  MoveL 2042 to (226.09, 430.21, -17.52) mm, rotated rx -180 ry 0 rz -11.91 deg; joints [26.659, -20.064, 61.919, -79.673, 100.73, 132.011]
  MoveL 2043 to (226.02, 430.34, -17.52) mm, rotated rx 180 ry 0 rz -11.91 deg; joints [26.655, -20.058, 61.906, -79.677, 100.728, 132.004]
  MoveL 2044 to (225.94, 430.47, -17.53) mm, rotated rx -180 ry 0 rz -11.91 deg; joints [26.652, -20.052, 61.893, -79.681, 100.727, 131.996]
  MoveL 2045 to (225.78, 430.71, -17.53) mm, rotated rx 180 ry 0 rz -11.91 deg; joints [26.644, -20.041, 61.871, -79.689, 100.723, 131.983]
  MoveL 2046 to (225.58, 430.96, -17.53) mm, rotated rx 180 ry 0 rz -11.91 deg; joints [26.635, -20.032, 61.851, -79.697, 100.718, 131.972]
  MoveL 2047 to (225.44, 431.1, -17.52) mm, rotated rx -180 ry 0 rz -11.91 deg; joints [26.629, -20.027, 61.84, -79.702, 100.715, 131.966]
  MoveL 2048 to (225.3, 431.23, -17.53) mm, rotated rx -180 ry 0 rz -11.91 deg; joints [26.623, -20.023, 61.833, -79.706, 100.712, 131.961]
  MoveL 2049 to (225.16, 431.34, -17.53) mm, rotated rx -180 ry 0 rz -11.91 deg; joints [26.618, -20.02, 61.827, -79.711, 100.708, 131.957]
  MoveL 2050 to (225.02, 431.44, -17.53) mm, rotated rx -180 ry 0 rz -11.91 deg; joints [26.612, -20.018, 61.822, -79.715, 100.705, 131.954]
  MoveL 2051 to (224.78, 431.59, -17.52) mm, rotated rx -180 ry 0 rz -11.91 deg; joints [26.604, -20.016, 61.818, -79.721, 100.699, 131.951]
  MoveL 2052 to (224.55, 431.71, -17.53) mm, rotated rx -180 ry 0 rz -11.91 deg; joints [26.596, -20.016, 61.818, -79.727, 100.693, 131.95]
  MoveL 2053 to (224.32, 431.8, -17.53) mm, rotated rx -180 ry 0 rz -11.91 deg; joints [26.588, -20.017, 61.821, -79.732, 100.687, 131.951]
  MoveL 2054 to (224.09, 431.88, -17.53) mm, rotated rx -180 ry 0 rz -11.91 deg; joints [26.581, -20.02, 61.827, -79.736, 100.681, 131.953]
  MoveL 2055 to (224.01, 431.9, -17.53) mm, rotated rx -180 ry 0 rz -11.91 deg; joints [26.579, -20.021, 61.829, -79.738, 100.679, 131.954]
  MoveL 2056 to (223.77, 431.95, -17.53) mm, rotated rx -180 ry 0 rz -11.91 deg; joints [26.571, -20.025, 61.839, -79.742, 100.673, 131.958]
  MoveL 2057 to (223.53, 431.98, -17.53) mm, rotated rx -180 ry 0 rz -11.91 deg; joints [26.564, -20.031, 61.851, -79.745, 100.666, 131.963]
  MoveL 2058 to (223.29, 431.99, -17.53) mm, rotated rx -180 ry 0 rz -11.91 deg; joints [26.557, -20.038, 61.866, -79.749, 100.66, 131.97]
  MoveL 2059 to (223.05, 431.99, -17.53) mm, rotated rx -180 ry 0 rz -11.91 deg; joints [26.551, -20.046, 61.883, -79.752, 100.653, 131.978]
  MoveL 2060 to (-164.9, 431.99, -17.52) mm, rotated rx -180 ry 0 rz -11.91 deg; joints [14.903, -28.534, 80.361, -87.324, 91.595, 141.007]
  MoveL 2061 to (-194.97, 431.99, -17.53) mm, rotated rx 180 ry 0 rz -11.91 deg; joints [13.93, -28.928, 81.241, -88.082, 90.978, 141.468]
  MoveL 2062 to (-195.47, 431.99, -17.53) mm, rotated rx 180 ry 0 rz -11.91 deg; joints [13.914, -28.934, 81.255, -88.094, 90.967, 141.475]
  Set speed (38.1 mm/s)
  MoveL 2063 to (-196.09, 432.77, -17.53) mm, rotated rx -180 ry 0 rz -11.91 deg; joints [13.888, -28.902, 81.184, -88.116, 90.952, 141.437]
  MoveL 2064 to (-195.65, 434.72, -17.52) mm, rotated rx 180 ry 0 rz -11.91 deg; joints [13.886, -28.795, 80.951, -88.119, 90.956, 141.311]
  MoveL 2065 to (-195.51, 435.34, -16.89) mm, rotated rx 180 ry 0 rz -11.91 deg; joints [13.886, -28.791, 80.884, -88.121, 90.957, 141.248]
  Set speed (100.0 mm/s)
  MoveL 2066 to (-195.51, 435.34, 34.52) mm, rotated rx 180 ry 0 rz -11.91 deg; joints [13.873, -31.158, 81.335, -88.164, 91.012, 139.332]
  MoveL 2067 to (-195.51, 435.34, 34.52) mm, rotated rx 180 ry 0 rz -11.91 deg; joints [13.873, -31.158, 81.335, -88.164, 91.012, 139.332]

--- program Machining (robot KUKA KR 30 HA) ---
  Smooth(15)
  Print: /'1001'
  Print: /''
  Print: /'Parallel1'
  Set speed (100.0 mm/s)
  Set Ref.: Frame 4
  Set Tool: rc90 spindle mm
  Show rc90 spindle mm
  MoveJ 1 to (194.72, 277.93, 99.72) mm, rotated rx -149.92 ry 0.28 rz 179.52 deg; joints [13.584, -45.402, 109.059, -165.249, 63.754, 203.812]
  MoveL 2 to (194.72, 277.93, 99.72) mm, rotated rx -149.92 ry 0.28 rz 179.52 deg; joints [13.584, -45.402, 109.059, -165.249, 63.754, 203.812]
  MoveL 3 to (194.72, 227.8, 13.19) mm, rotated rx -149.92 ry 0.28 rz 179.52 deg; joints [15.532, -40.122, 107.271, -163.55, 67.335, 203.986]
  MoveL 4 to (194.72, 227.8, 13.19) mm, rotated rx -149.92 ry 0.28 rz 179.52 deg; joints [15.532, -40.122, 107.271, -163.55, 67.335, 203.986]
  Set speed (100.0 mm/s)
  MoveL 5 to (194.72, 218.79, -2.36) mm, rotated rx -149.92 ry 0.28 rz 179.52 deg; joints [15.878, -39.152, 106.869, -163.244, 67.917, 204.023]
  Set speed (16.7 mm/s)
  MoveL 6 to (194.72, 209.92, -17.68) mm, rotated rx -149.92 ry 0.28 rz 179.52 deg; joints [16.219, -38.193, 106.45, -162.942, 68.471, 204.061]
  MoveL 7 to (193.72, 209.42, -18.55) mm, rotated rx -149.92 ry 0.28 rz 179.52 deg; joints [16.249, -38.173, 106.512, -162.919, 68.552, 204.075]
  MoveL 8 to (193.59, 214.43, -9.89) mm, rotated rx -149.92 ry 0.28 rz 179.52 deg; joints [16.058, -38.721, 106.764, -163.089, 68.248, 204.055]
  MoveL 9 to (193.59, 214.44, -9.88) mm, rotated rx -149.92 ry 0.28 rz 179.52 deg; joints [16.058, -38.722, 106.764, -163.089, 68.248, 204.055]
  Set speed (100.0 mm/s)
  MoveL 10 to (193.59, 222.79, 4.53) mm, rotated rx -149.92 ry 0.28 rz 179.52 deg; joints [15.737, -39.624, 107.148, -163.373, 67.718, 204.02]
  MoveL 11 to (194.72, 224.52, 3.53) mm, rotated rx -149.92 ry 0.28 rz 179.52 deg; joints [15.659, -39.543, 107.081, -163.458, 67.722, 204.054]
  MoveL 12 to (194.72, 217.03, -9.4) mm, rotated rx -149.92 ry 0.28 rz 179.52 deg; joints [15.947, -38.735, 106.737, -163.203, 68.198, 204.085]
  Set speed (16.7 mm/s)
  MoveL 13 to (194.72, 211.65, -18.68) mm, rotated rx -149.92 ry 0.28 rz 179.52 deg; joints [16.154, -38.152, 106.48, -163.02, 68.531, 204.108]
  MoveC 14 to (194.43, 211.3, -19.3) mm, rotated rx -149.92 ry 0.28 rz 179.52 deg; joints [16.17, -38.124, 106.488, -163.006, 68.568, 204.113] to (193.72, 211.15, -19.55) mm, rotated rx -149.92 ry 0.28 rz 179.52 deg; joints [16.184, -38.133, 106.542, -162.997, 68.613, 204.122]
  MoveL 15 to (193.72, 211.15, -19.55) mm, rotated rx -149.92 ry 0.28 rz 179.52 deg; joints [16.184, -38.133, 106.542, -162.997, 68.613, 204.122]
  MoveL 16 to (193.49, 216.16, -10.9) mm, rotated rx -149.92 ry 0.28 rz 179.52 deg; joints [15.994, -38.685, 106.803, -163.166, 68.314, 204.104]
  MoveL 17 to (191.2, 216.16, -10.9) mm, rotated rx -149.92 ry 0.28 rz 179.52 deg; joints [16.019, -38.765, 107.001, -163.153, 68.429, 204.131]
  MoveC 18 to (190.5, 216.31, -10.64) mm, rotated rx -149.92 ry 0.28 rz 179.52 deg; joints [16.021, -38.806, 107.069, -163.154, 68.455, 204.138] to (190.2, 216.66, -10.03) mm, rotated rx -149.92 ry 0.28 rz 179.52 deg; joints [16.011, -38.855, 107.111, -163.164, 68.448, 204.14]
  MoveL 19 to (190.2, 216.66, -10.03) mm, rotated rx -149.92 ry 0.28 rz 179.52 deg; joints [16.011, -38.855, 107.111, -163.164, 68.448, 204.14]
  Set speed (100.0 mm/s)
  MoveL 20 to (190.2, 224.52, 3.53) mm, rotated rx -149.92 ry 0.28 rz 179.52 deg; joints [15.708, -39.705, 107.472, -163.432, 67.947, 204.106]
  MoveL 21 to (-191.54, 222.79, 4.53) mm, rotated rx -149.92 ry 0.28 rz 179.52 deg; joints [21.283, -50.457, 136.898, -159.048, 86.021, 209.028]
  MoveL 22 to (-191.54, 219.49, -1.15) mm, rotated rx -149.92 ry 0.28 rz 179.52 deg; joints [21.448, -49.971, 136.724, -158.89, 86.316, 209.131]
  Set speed (16.7 mm/s)
  MoveL 23 to (-191.54, 214.63, -9.56) mm, rotated rx -149.92 ry 0.28 rz 179.52 deg; joints [21.69, -49.254, 136.461, -158.658, 86.744, 209.284]
  MoveL 24 to (-191.93, 214.43, -9.89) mm, rotated rx -149.92 ry 0.28 rz 179.52 deg; joints [21.707, -49.232, 136.477, -158.641, 86.78, 209.297]
  MoveL 25 to (-192.68, 214.43, -9.89) mm, rotated rx -149.92 ry 0.28 rz 179.52 deg; joints [21.722, -49.246, 136.529, -158.627, 86.815, 209.31]
  MoveL 26 to (-192.7, 209.42, -18.55) mm, rotated rx -149.92 ry 0.28 rz 179.52 deg; joints [21.971, -48.509, 136.25, -158.387, 87.245, 209.468]
  MoveL 27 to (-193.07, 211.15, -19.55) mm, rotated rx -149.92 ry 0.28 rz 179.52 deg; joints [21.894, -48.445, 136.307, -158.465, 87.357, 209.515]
  MoveL 28 to (-193.07, 216.16, -10.9) mm, rotated rx -149.92 ry 0.28 rz 179.52 deg; joints [21.645, -49.182, 136.587, -158.707, 86.927, 209.358]
  MoveL 29 to (-189.43, 216.16, -10.9) mm, rotated rx -149.92 ry 0.28 rz 179.52 deg; joints [21.574, -49.115, 136.335, -158.774, 86.753, 209.294]
  MoveL 30 to (-188.93, 216.41, -10.46) mm, rotated rx -149.92 ry 0.28 rz 179.52 deg; joints [21.552, -49.143, 136.314, -158.795, 86.708, 209.277]
  MoveC 31 to (-189.34, 217.09, -9.63) mm, rotated rx -149.92 ry 0.28 rz 179.52 deg; joints [21.527, -49.223, 136.374, -158.82, 86.689, 209.271] to (-190.32, 217.64, -9.44) mm, rotated rx -149.92 ry 0.28 rz 179.52 deg; joints [21.519, -49.26, 136.461, -158.829, 86.735, 209.289]
  MoveL 32 to (-190.32, 217.64, -9.44) mm, rotated rx -149.92 ry 0.28 rz 179.52 deg; joints [21.519, -49.26, 136.461, -158.829, 86.735, 209.289]
  MoveL 33 to (-192.56, 218.42, -9.89) mm, rotated rx -149.92 ry 0.28 rz 179.52 deg; joints [21.525, -49.27, 136.63, -158.826, 86.884, 209.347]
  MoveC 34 to (-193.55, 218.53, -10.47) mm, rotated rx -149.92 ry 0.28 rz 179.52 deg; joints [21.538, -49.242, 136.692, -158.815, 86.968, 209.379] to (-193.96, 218.14, -11.47) mm, rotated rx -149.92 ry 0.28 rz 179.52 deg; joints [21.566, -49.165, 136.694, -158.788, 87.042, 209.406]
  MoveL 35 to (-193.96, 218.14, -11.47) mm, rotated rx -149.92 ry 0.28 rz 179.52 deg; joints [21.566, -49.165, 136.694, -158.788, 87.042, 209.406]
  MoveL 36 to (-193.96, 213.13, -20.12) mm, rotated rx -149.92 ry 0.28 rz 179.52 deg; joints [21.815, -48.426, 136.413, -158.546, 87.472, 209.564]
  MoveL 37 to (-193.46, 212.88, -20.55) mm, rotated rx -149.92 ry 0.28 rz 179.52 deg; joints [21.818, -48.381, 136.364, -158.544, 87.469, 209.563]
  MoveL 38 to (-193.43, 217.89, -11.9) mm, rotated rx -149.92 ry 0.28 rz 179.52 deg; joints [21.568, -49.118, 136.644, -158.786, 87.038, 209.405]
  MoveL 39 to (193.49, 217.89, -11.9) mm, rotated rx -149.92 ry 0.28 rz 179.52 deg; joints [15.929, -38.644, 106.833, -163.244, 68.375, 204.151]
  MoveL 40 to (193.72, 212.88, -20.55) mm, rotated rx -149.92 ry 0.28 rz 179.52 deg; joints [16.119, -38.092, 106.572, -163.074, 68.673, 204.169]
  MoveL 41 to (193.72, 214.61, -21.55) mm, rotated rx -149.92 ry 0.28 rz 179.52 deg; joints [16.054, -38.052, 106.601, -163.152, 68.733, 204.215]
  MoveL 42 to (193.49, 219.62, -12.9) mm, rotated rx -149.92 ry 0.28 rz 179.52 deg; joints [15.864, -38.604, 106.863, -163.322, 68.435, 204.197]
  MoveL 43 to (-193.72, 219.62, -12.9) mm, rotated rx -149.92 ry 0.28 rz 179.52 deg; joints [21.489, -49.053, 136.695, -158.867, 87.146, 209.45]
  MoveL 44 to (-193.74, 214.61, -21.55) mm, rotated rx -149.92 ry 0.28 rz 179.52 deg; joints [21.74, -48.314, 136.415, -158.624, 87.576, 209.608]
  MoveL 45 to (-193.31, 216.34, -22.56) mm, rotated rx -149.92 ry 0.28 rz 179.52 deg; joints [21.647, -48.236, 136.416, -158.718, 87.649, 209.639]
  MoveL 46 to (-193.31, 221.35, -13.9) mm, rotated rx -149.92 ry 0.28 rz 179.52 deg; joints [21.397, -48.974, 136.697, -158.961, 87.22, 209.483]
  MoveL 47 to (193.28, 221.35, -13.9) mm, rotated rx -149.92 ry 0.28 rz 179.52 deg; joints [15.8, -38.57, 106.91, -163.399, 68.506, 204.246]
  MoveL 48 to (193.31, 216.34, -22.56) mm, rotated rx -149.92 ry 0.28 rz 179.52 deg; joints [15.993, -38.025, 106.666, -163.227, 68.814, 204.266]
  MoveL 49 to (191.75, 218.07, -23.56) mm, rotated rx -149.92 ry 0.28 rz 179.52 deg; joints [15.945, -38.038, 106.83, -163.295, 68.953, 204.331]
  MoveL 50 to (191.68, 223.08, -14.91) mm, rotated rx -149.92 ry 0.28 rz 179.52 deg; joints [15.752, -38.585, 107.077, -163.467, 68.646, 204.311]
  MoveL 51 to (-191.75, 223.08, -14.91) mm, rotated rx -149.92 ry 0.28 rz 179.52 deg; joints [21.282, -48.875, 136.619, -159.076, 87.238, 209.495]
  MoveL 52 to (-191.75, 218.07, -23.56) mm, rotated rx -149.92 ry 0.28 rz 179.52 deg; joints [21.532, -48.137, 136.337, -158.833, 87.667, 209.65]
  MoveC 53 to (-192.46, 218.22, -23.31) mm, rotated rx -149.92 ry 0.28 rz 179.52 deg; joints [21.539, -48.171, 136.395, -158.827, 87.689, 209.658] to (-192.75, 218.57, -22.69) mm, rotated rx -149.92 ry 0.28 rz 179.52 deg; joints [21.527, -48.228, 136.435, -158.839, 87.673, 209.653]
  MoveL 54 to (-192.75, 218.57, -22.69) mm, rotated rx -149.92 ry 0.28 rz 179.52 deg; joints [21.527, -48.228, 136.435, -158.839, 87.673, 209.653]
  Set speed (100.0 mm/s)
  MoveL 55 to (-192.75, 236.46, 8.18) mm, rotated rx -149.92 ry 0.28 rz 179.52 deg; joints [20.63, -50.873, 137.4, -159.704, 86.088, 209.096]
  Print: /'Parallel2'
  Set speed (100.0 mm/s)
  MoveL 56 to (-122.87, -170.47, 35.88) mm, rotated rx -149.92 ry 0.28 rz 179.52 deg; joints [36.036, -45.854, 117.438, -142.779, 74.483, 199.283]
  MoveL 57 to (-122.87, -192.28, -1.78) mm, rotated rx -149.92 ry 0.28 rz 179.52 deg; joints [36.803, -43.103, 115.933, -142.202, 75.615, 199.876]
  Set speed (16.7 mm/s)
  MoveL 58 to (-122.87, -206.58, -26.46) mm, rotated rx -149.92 ry 0.28 rz 179.52 deg; joints [37.298, -41.303, 114.871, -141.813, 76.284, 200.228]
  MoveC 59 to (-122.57, -206.94, -27.07) mm, rotated rx -149.92 ry 0.28 rz 179.52 deg; joints [37.303, -41.25, 114.824, -141.809, 76.289, 200.23] to (-121.87, -207.08, -27.32) mm, rotated rx -149.92 ry 0.28 rz 179.52 deg; joints [37.29, -41.214, 114.765, -141.819, 76.27, 200.219]
  MoveL 60 to (-121.87, -207.08, -27.32) mm, rotated rx -149.92 ry 0.28 rz 179.52 deg; joints [37.29, -41.214, 114.765, -141.819, 76.27, 200.219]
  MoveL 61 to (-121.78, -193.28, -3.5) mm, rotated rx -149.92 ry 0.28 rz 179.52 deg; joints [36.81, -42.948, 115.788, -142.196, 75.623, 199.88]
  MoveL 62 to (189.07, -193.28, -3.5) mm, rotated rx -149.92 ry 0.28 rz 179.52 deg; joints [30.162, -32.815, 91.718, -146.035, 62.74, 193.528]
  MoveL 63 to (189.08, -207.08, -27.32) mm, rotated rx -149.92 ry 0.28 rz 179.52 deg; joints [30.593, -31.289, 90.675, -145.71, 63.263, 193.626]
  MoveL 64 to (192.38, -208.45, -26.53) mm, rotated rx -149.92 ry 0.28 rz 179.52 deg; joints [30.575, -31.169, 90.316, -145.661, 63.06, 193.483]
  MoveL 65 to (193.72, -211.41, -24.82) mm, rotated rx -149.92 ry 0.28 rz 179.52 deg; joints [30.64, -31.137, 90.062, -145.528, 62.896, 193.312]
  MoveL 66 to (193.72, -197.6, -1) mm, rotated rx -149.92 ry 0.28 rz 179.52 deg; joints [30.21, -32.66, 91.107, -145.851, 62.376, 193.216]
  MoveL 67 to (-126.28, -197.6, -1) mm, rotated rx -149.92 ry 0.28 rz 179.52 deg; joints [37.07, -43.141, 115.904, -141.92, 75.61, 199.769]
  MoveL 68 to (-126.51, -211.41, -24.82) mm, rotated rx -149.92 ry 0.28 rz 179.52 deg; joints [37.552, -41.408, 114.892, -141.543, 76.263, 200.116]
  MoveL 69 to (-126.14, -213.57, -23.57) mm, rotated rx -149.92 ry 0.28 rz 179.52 deg; joints [37.614, -41.435, 114.773, -141.458, 76.16, 200.008]
  MoveL 70 to (-125.68, -215.73, -22.32) mm, rotated rx -149.92 ry 0.28 rz 179.52 deg; joints [37.673, -41.459, 114.648, -141.375, 76.054, 199.898]
  MoveL 71 to (-125.64, -207.44, -8.02) mm, rotated rx -149.92 ry 0.28 rz 179.52 deg; joints [37.388, -42.5, 115.268, -141.598, 75.672, 199.695]
  MoveL 72 to (-121.57, -207.44, -8.02) mm, rotated rx -149.92 ry 0.28 rz 179.52 deg; joints [37.284, -42.393, 114.993, -141.677, 75.522, 199.613]
  MoveL 73 to (-121.42, -201.93, 1.51) mm, rotated rx -149.92 ry 0.28 rz 179.52 deg; joints [37.09, -43.082, 115.386, -141.826, 75.253, 199.471]
  MoveL 74 to (188.78, -201.93, 1.51) mm, rotated rx -149.92 ry 0.28 rz 179.52 deg; joints [30.43, -32.885, 91.353, -145.62, 62.458, 193.123]
  MoveL 75 to (188.9, -207.44, -8.02) mm, rotated rx -149.92 ry 0.28 rz 179.52 deg; joints [30.6, -32.273, 90.933, -145.494, 62.667, 193.163]
  MoveL 76 to (193.72, -207.44, -8.02) mm, rotated rx -149.92 ry 0.28 rz 179.52 deg; joints [30.513, -32.081, 90.5, -145.516, 62.442, 193.051]
  MoveL 77 to (193.72, -215.73, -22.32) mm, rotated rx -149.92 ry 0.28 rz 179.52 deg; joints [30.77, -31.165, 89.865, -145.323, 62.749, 193.106]
  MoveL 78 to (193.72, -217.89, -21.07) mm, rotated rx -149.92 ry 0.28 rz 179.52 deg; joints [30.834, -31.179, 89.766, -145.22, 62.676, 193.003]
  MoveL 79 to (193.7, -220.05, -19.82) mm, rotated rx -149.92 ry 0.28 rz 179.52 deg; joints [30.899, -31.194, 89.669, -145.117, 62.603, 192.899]
  MoveL 80 to (193.7, -211.76, -5.52) mm, rotated rx -149.92 ry 0.28 rz 179.52 deg; joints [30.643, -32.109, 90.303, -145.309, 62.296, 192.843]
  MoveL 81 to (-124.73, -211.76, -5.52) mm, rotated rx -149.92 ry 0.28 rz 179.52 deg; joints [37.508, -42.547, 115.016, -141.429, 75.461, 199.475]
  MoveL 82 to (-124.77, -220.05, -19.82) mm, rotated rx -149.92 ry 0.28 rz 179.52 deg; joints [37.791, -41.507, 114.398, -141.208, 75.842, 199.678]
  MoveC 83 to (-125.47, -219.9, -19.56) mm, rotated rx -149.92 ry 0.28 rz 179.52 deg; joints [37.805, -41.544, 114.456, -141.198, 75.862, 199.689] to (-125.77, -219.55, -18.95) mm, rotated rx -149.92 ry 0.28 rz 179.52 deg; joints [37.8, -41.596, 114.503, -141.202, 75.857, 199.687]
  MoveL 84 to (-125.77, -219.55, -18.95) mm, rotated rx -149.92 ry 0.28 rz 179.52 deg; joints [37.8, -41.596, 114.503, -141.202, 75.857, 199.687]
  Set speed (100.0 mm/s)
  MoveL 85 to (-125.77, -183.44, 43.39) mm, rotated rx -149.92 ry 0.28 rz 179.52 deg; joints [36.551, -46.139, 117.057, -142.14, 74.056, 198.725]
  Print: /'Contour6'
  Set speed (100.0 mm/s)
  MoveL 86 to (-194.89, 224.1, 15) mm, rotated rx -180 ry 0 rz 179.9 deg; joints [27.663, -53.009, 133.443, -151.936, 80.607, 175.728]
  MoveL 87 to (-194.89, 224.1, 1.16) mm, rotated rx 180 ry 0 rz 179.9 deg; joints [27.67, -51.959, 133.305, -151.996, 81.413, 176.161]
  Set speed (5.6 mm/s)
  MoveL 88 to (-194.89, 224.1, -5) mm, rotated rx 180 ry 0 rz 179.9 deg; joints [27.674, -51.49, 133.238, -152.021, 81.768, 176.351]
  MoveC 89 to (-194.65, 223.92, -5.71) mm, rotated rx 180 ry 0 rz 179.9 deg; joints [27.676, -51.428, 133.208, -152.02, 81.796, 176.366] to (-194.08, 223.5, -6) mm, rotated rx -180 ry 0 rz 179.9 deg; joints [27.682, -51.388, 133.151, -152.013, 81.782, 176.357]
  Set speed (16.7 mm/s)
  MoveL 90 to (-190.41, 220.78, -6) mm, rotated rx 180 ry 0 rz 179.9 deg; joints [27.717, -51.27, 132.805, -151.963, 81.583, 176.244]
  MoveL 91 to (-190.31, 219.26, -6) mm, rotated rx -180 ry 0 rz 179.9 deg; joints [27.782, -51.249, 132.743, -151.894, 81.551, 176.216]
  MoveL 92 to (-190.6, 218.98, -6) mm, rotated rx -180 ry 0 rz 179.9 deg; joints [27.801, -51.253, 132.753, -151.876, 81.557, 176.217]
  MoveL 93 to (-190.82, 218.73, -6) mm, rotated rx -180 ry 0 rz 179.9 deg; joints [27.817, -51.256, 132.759, -151.859, 81.562, 176.216]
  MoveL 94 to (-191.02, 218.47, -6) mm, rotated rx -180 ry 0 rz 179.9 deg; joints [27.833, -51.257, 132.764, -151.843, 81.565, 176.215]
  MoveL 95 to (-191.23, 218.16, -6) mm, rotated rx 180 ry 0 rz 179.9 deg; joints [27.852, -51.259, 132.767, -151.825, 81.568, 176.214]
  MoveL 96 to (-191.4, 217.86, -6) mm, rotated rx 180 ry 0 rz 179.9 deg; joints [27.869, -51.259, 132.767, -151.807, 81.57, 176.212]
  MoveL 97 to (-191.55, 217.55, -6) mm, rotated rx 180 ry 0 rz 179.9 deg; joints [27.886, -51.259, 132.766, -151.79, 81.57, 176.209]
  MoveL 98 to (-191.68, 217.24, -6) mm, rotated rx 180 ry 0 rz 179.9 deg; joints [27.903, -51.258, 132.764, -151.773, 81.569, 176.206]
  MoveL 99 to (-191.78, 216.94, -6) mm, rotated rx 180 ry 0 rz 179.9 deg; joints [27.919, -51.257, 132.76, -151.757, 81.568, 176.202]
  MoveL 100 to (-191.86, 216.63, -6) mm, rotated rx 180 ry 0 rz 179.9 deg; joints [27.934, -51.255, 132.754, -151.741, 81.565, 176.198]
  MoveL 101 to (-191.91, 216.32, -6) mm, rotated rx 180 ry 0 rz 179.9 deg; joints [27.949, -51.253, 132.747, -151.726, 81.562, 176.194]
  MoveL 102 to (-191.95, 216.02, -6) mm, rotated rx -180 ry 0 rz 179.9 deg; joints [27.963, -51.251, 132.738, -151.711, 81.558, 176.189]
  MoveL 103 to (-191.97, 215.71, -6) mm, rotated rx 180 ry 0 rz 179.9 deg; joints [27.977, -51.248, 132.729, -151.696, 81.553, 176.184]
  MoveL 104 to (-191.98, 215.4, -6) mm, rotated rx 180 ry 0 rz 179.9 deg; joints [27.991, -51.244, 132.718, -151.682, 81.548, 176.179]
  MoveL 105 to (-191.98, 213.56, -6) mm, rotated rx -180 ry 0 rz 179.9 deg; joints [28.072, -51.222, 132.651, -151.597, 81.514, 176.147]
  MoveL 106 to (-191.97, 212.33, -6) mm, rotated rx 180 ry 0 rz 179.9 deg; joints [28.126, -51.208, 132.606, -151.54, 81.491, 176.125]
  MoveL 107 to (-191.94, 212.03, -6) mm, rotated rx 180 ry 0 rz 179.9 deg; joints [28.139, -51.203, 132.593, -151.527, 81.484, 176.119]
  MoveL 108 to (-191.89, 211.72, -6) mm, rotated rx 180 ry 0 rz 179.9 deg; joints [28.151, -51.199, 132.579, -151.514, 81.477, 176.113]
  MoveL 109 to (-126.45, -201.29, -6) mm, rotated rx -180 ry 0 rz 179.9 deg; joints [41.507, -41.984, 108.551, -135.769, 71.778, 164.105]
  MoveL 110 to (-126.38, -201.66, -6) mm, rotated rx -180 ry 0 rz 179.9 deg; joints [41.516, -41.973, 108.524, -135.756, 71.769, 164.091]
  MoveL 111 to (-126.27, -202.03, -6) mm, rotated rx 180 ry 0 rz 179.9 deg; joints [41.524, -41.96, 108.495, -135.744, 71.759, 164.076]
  MoveL 112 to (-126.2, -202.24, -6) mm, rotated rx -180 ry 0 rz 179.9 deg; joints [41.529, -41.953, 108.478, -135.737, 71.753, 164.068]
  MoveL 113 to (-126.11, -202.46, -6) mm, rotated rx -180 ry 0 rz 179.9 deg; joints [41.533, -41.945, 108.459, -135.73, 71.747, 164.058]
  MoveL 114 to (-126.02, -202.67, -6) mm, rotated rx -180 ry 0 rz 179.9 deg; joints [41.536, -41.937, 108.44, -135.724, 71.74, 164.049]
  MoveL 115 to (-125.91, -202.89, -6) mm, rotated rx -180 ry 0 rz 179.9 deg; joints [41.54, -41.929, 108.42, -135.718, 71.733, 164.04]
  MoveL 116 to (-125.78, -203.1, -6) mm, rotated rx 180 ry 0 rz 179.9 deg; joints [41.543, -41.92, 108.399, -135.712, 71.725, 164.03]
  MoveL 117 to (-125.64, -203.31, -6) mm, rotated rx -180 ry 0 rz 179.9 deg; joints [41.546, -41.91, 108.377, -135.706, 71.717, 164.02]
  MoveL 118 to (-125.49, -203.53, -6) mm, rotated rx 180 ry 0 rz 179.9 deg; joints [41.548, -41.901, 108.354, -135.701, 71.708, 164.009]
  MoveL 119 to (-125.32, -203.74, -6) mm, rotated rx 180 ry 0 rz 179.9 deg; joints [41.55, -41.89, 108.33, -135.696, 71.698, 163.999]
  MoveL 120 to (-125.14, -203.94, -6) mm, rotated rx -180 ry 0 rz 179.9 deg; joints [41.551, -41.88, 108.306, -135.691, 71.689, 163.988]
  MoveL 121 to (-124.94, -204.13, -6) mm, rotated rx 180 ry 0 rz 179.9 deg; joints [41.552, -41.87, 108.281, -135.688, 71.679, 163.978]
  MoveL 122 to (-124.76, -204.3, -6) mm, rotated rx -180 ry 0 rz 179.9 deg; joints [41.552, -41.86, 108.259, -135.685, 71.67, 163.968]
  MoveL 123 to (-124.57, -204.45, -6) mm, rotated rx 180 ry 0 rz 179.9 deg; joints [41.551, -41.851, 108.237, -135.682, 71.661, 163.959]
  MoveL 124 to (-124.2, -204.72, -6) mm, rotated rx 180 ry 0 rz 179.9 deg; joints [41.549, -41.833, 108.197, -135.679, 71.644, 163.943]
  MoveL 125 to (-123.82, -204.93, -6) mm, rotated rx 180 ry 0 rz 179.9 deg; joints [41.546, -41.817, 108.159, -135.677, 71.627, 163.928]
  MoveL 126 to (-123.52, -205.08, -6) mm, rotated rx -180 ry 0 rz 179.9 deg; joints [41.542, -41.805, 108.129, -135.677, 71.614, 163.917]
  MoveL 127 to (-123.21, -205.2, -6) mm, rotated rx -180 ry 0 rz 179.9 deg; joints [41.537, -41.793, 108.102, -135.678, 71.601, 163.906]
  MoveL 128 to (-122.9, -205.3, -6) mm, rotated rx 180 ry 0 rz 179.9 deg; joints [41.532, -41.781, 108.075, -135.68, 71.589, 163.897]
  MoveL 129 to (-122.6, -205.38, -6) mm, rotated rx -180 ry 0 rz 179.9 deg; joints [41.526, -41.77, 108.05, -135.682, 71.577, 163.888]
  MoveL 130 to (-122.29, -205.44, -6) mm, rotated rx 180 ry 0 rz 179.9 deg; joints [41.52, -41.76, 108.026, -135.685, 71.566, 163.88]
  MoveL 131 to (-121.98, -205.47, -6) mm, rotated rx 180 ry 0 rz 179.9 deg; joints [41.513, -41.75, 108.003, -135.689, 71.555, 163.872]
  MoveL 132 to (-121.37, -205.5, -6) mm, rotated rx 180 ry 0 rz 179.9 deg; joints [41.498, -41.731, 107.96, -135.699, 71.533, 163.859]
  MoveL 133 to (182.67, -205.5, -6) mm, rotated rx -180 ry 0 rz 179.9 deg; joints [34.628, -30.981, 84.081, -138.767, 59.535, 156.897]
  MoveL 134 to (188.8, -205.49, -6) mm, rotated rx -180 ry 0 rz 179.9 deg; joints [34.51, -30.717, 83.511, -138.774, 59.257, 156.724]
  MoveL 135 to (189.1, -205.48, -6) mm, rotated rx 180 ry 0 rz 179.9 deg; joints [34.503, -30.704, 83.483, -138.775, 59.243, 156.716]
  MoveL 136 to (189.41, -205.45, -6) mm, rotated rx -180 ry 0 rz 179.9 deg; joints [34.497, -30.692, 83.457, -138.776, 59.23, 156.709]
  MoveL 137 to (189.72, -205.4, -6) mm, rotated rx 180 ry 0 rz 179.9 deg; joints [34.489, -30.68, 83.431, -138.779, 59.217, 156.702]
  MoveL 138 to (190.02, -205.32, -6) mm, rotated rx 180 ry 0 rz 179.9 deg; joints [34.481, -30.669, 83.407, -138.782, 59.204, 156.697]
  MoveL 139 to (190.26, -205.25, -6) mm, rotated rx 180 ry 0 rz 179.9 deg; joints [34.475, -30.661, 83.39, -138.785, 59.195, 156.693]
  MoveL 140 to (190.64, -205.11, -6) mm, rotated rx -180 ry 0 rz 179.9 deg; joints [34.464, -30.649, 83.363, -138.792, 59.179, 156.688]
  MoveL 141 to (190.94, -204.97, -6) mm, rotated rx 180 ry 0 rz 179.9 deg; joints [34.454, -30.64, 83.344, -138.798, 59.168, 156.685]
  MoveL 142 to (191.25, -204.81, -6) mm, rotated rx -180 ry 0 rz 179.9 deg; joints [34.444, -30.631, 83.326, -138.805, 59.156, 156.683]
  MoveL 143 to (191.56, -204.61, -6) mm, rotated rx 180 ry 0 rz 179.9 deg; joints [34.432, -30.623, 83.309, -138.814, 59.145, 156.683]
  MoveL 144 to (191.86, -204.39, -6) mm, rotated rx -180 ry 0 rz 179.9 deg; joints [34.42, -30.617, 83.295, -138.824, 59.135, 156.684]
  MoveL 145 to (192.17, -204.12, -6) mm, rotated rx 180 ry 0 rz 179.9 deg; joints [34.407, -30.611, 83.284, -138.836, 59.125, 156.686]
  MoveL 146 to (192.33, -203.96, -6) mm, rotated rx -180 ry 0 rz 179.9 deg; joints [34.399, -30.609, 83.279, -138.843, 59.12, 156.688]
  MoveL 147 to (192.48, -203.8, -6) mm, rotated rx 180 ry 0 rz 179.9 deg; joints [34.392, -30.607, 83.276, -138.85, 59.116, 156.691]
  MoveL 148 to (192.52, -203.74, -6) mm, rotated rx 180 ry 0 rz 179.9 deg; joints [34.389, -30.607, 83.275, -138.853, 59.115, 156.692]
  MoveL 149 to (192.77, -203.44, -6) mm, rotated rx 180 ry 0 rz 179.9 deg; joints [34.376, -30.605, 83.272, -138.866, 59.108, 156.698]
  MoveL 150 to (192.97, -203.13, -6) mm, rotated rx 180 ry 0 rz 179.9 deg; joints [34.364, -30.605, 83.272, -138.88, 59.104, 156.705]
  MoveL 151 to (193.15, -202.82, -6) mm, rotated rx 180 ry 0 rz 179.9 deg; joints [34.352, -30.607, 83.275, -138.893, 59.1, 156.712]
  MoveL 152 to (193.3, -202.51, -6) mm, rotated rx -180 ry 0 rz 179.9 deg; joints [34.34, -30.609, 83.281, -138.907, 59.098, 156.721]
  MoveL 153 to (193.42, -202.21, -6) mm, rotated rx 180 ry 0 rz 179.9 deg; joints [34.329, -30.613, 83.289, -138.92, 59.097, 156.73]
  MoveL 154 to (193.52, -201.9, -6) mm, rotated rx -180 ry 0 rz 179.9 deg; joints [34.319, -30.617, 83.3, -138.934, 59.097, 156.74]
  MoveL 155 to (193.6, -201.59, -6) mm, rotated rx -180 ry 0 rz 179.9 deg; joints [34.309, -30.623, 83.312, -138.947, 59.099, 156.751]
  MoveL 156 to (193.66, -201.29, -6) mm, rotated rx 180 ry 0 rz 179.9 deg; joints [34.299, -30.629, 83.326, -138.961, 59.101, 156.762]
  MoveL 157 to (193.7, -200.98, -6) mm, rotated rx 180 ry 0 rz 179.9 deg; joints [34.29, -30.636, 83.342, -138.974, 59.103, 156.774]
  MoveL 158 to (193.72, -200.67, -6) mm, rotated rx 180 ry 0 rz 179.9 deg; joints [34.281, -30.644, 83.36, -138.987, 59.107, 156.786]
  MoveL 159 to (193.72, -200.06, -6) mm, rotated rx 180 ry 0 rz 179.9 deg; joints [34.264, -30.662, 83.399, -139.014, 59.116, 156.811]
  MoveL 160 to (193.72, 215.4, -6) mm, rotated rx -180 ry 0 rz 179.9 deg; joints [21.032, -39.388, 103.249, -156.64, 64.802, 170.151]
  MoveL 161 to (193.72, 215.71, -6) mm, rotated rx -180 ry 0 rz 179.9 deg; joints [21.021, -39.393, 103.26, -156.653, 64.805, 170.158]
  MoveL 162 to (193.7, 216.02, -6) mm, rotated rx -180 ry 0 rz 179.9 deg; joints [21.01, -39.398, 103.272, -156.666, 64.81, 170.166]
  MoveL 163 to (193.66, 216.32, -6) mm, rotated rx -180 ry 0 rz 179.9 deg; joints [21, -39.404, 103.286, -156.678, 64.815, 170.174]
  MoveL 164 to (193.6, 216.63, -6) mm, rotated rx -180 ry 0 rz 179.9 deg; joints [20.99, -39.41, 103.301, -156.691, 64.821, 170.183]
  MoveL 165 to (193.52, 216.94, -6) mm, rotated rx -180 ry 0 rz 179.9 deg; joints [20.98, -39.418, 103.318, -156.704, 64.829, 170.191]
  MoveL 166 to (193.42, 217.24, -6) mm, rotated rx 180 ry 0 rz 179.9 deg; joints [20.97, -39.426, 103.337, -156.716, 64.837, 170.2]
  MoveL 167 to (193.3, 217.55, -6) mm, rotated rx -180 ry 0 rz 179.9 deg; joints [20.961, -39.435, 103.358, -156.728, 64.846, 170.21]
  MoveL 168 to (193.15, 217.86, -6) mm, rotated rx 180 ry 0 rz 179.9 deg; joints [20.952, -39.445, 103.381, -156.74, 64.857, 170.22]
  MoveL 169 to (192.97, 218.16, -6) mm, rotated rx -180 ry 0 rz 179.9 deg; joints [20.943, -39.456, 103.407, -156.752, 64.869, 170.23]
  MoveL 170 to (192.77, 218.47, -6) mm, rotated rx -180 ry 0 rz 179.9 deg; joints [20.935, -39.468, 103.435, -156.764, 64.882, 170.24]
  MoveL 171 to (192.63, 218.65, -6) mm, rotated rx 180 ry 0 rz 179.9 deg; joints [20.931, -39.476, 103.453, -156.771, 64.891, 170.247]
  MoveL 172 to (192.48, 218.84, -6) mm, rotated rx -180 ry 0 rz 179.9 deg; joints [20.926, -39.484, 103.472, -156.778, 64.9, 170.254]
  MoveL 173 to (192.33, 219, -6) mm, rotated rx 180 ry 0 rz 179.9 deg; joints [20.922, -39.492, 103.491, -156.784, 64.909, 170.26]
  MoveL 174 to (192.17, 219.16, -6) mm, rotated rx -180 ry 0 rz 179.9 deg; joints [20.919, -39.5, 103.51, -156.79, 64.918, 170.266]
  MoveL 175 to (191.86, 219.42, -6) mm, rotated rx 180 ry 0 rz 179.9 deg; joints [20.914, -39.516, 103.545, -156.799, 64.936, 170.277]
  MoveL 176 to (191.56, 219.65, -6) mm, rotated rx -180 ry 0 rz 179.9 deg; joints [20.91, -39.531, 103.58, -156.807, 64.953, 170.287]
  MoveL 177 to (191.25, 219.85, -6) mm, rotated rx 180 ry 0 rz 179.9 deg; joints [20.907, -39.545, 103.613, -156.814, 64.97, 170.297]
  MoveL 178 to (190.94, 220.01, -6) mm, rotated rx 180 ry 0 rz 179.9 deg; joints [20.905, -39.559, 103.645, -156.819, 64.986, 170.305]
  MoveL 179 to (190.64, 220.15, -6) mm, rotated rx -180 ry 0 rz 179.9 deg; joints [20.904, -39.572, 103.676, -156.823, 65.002, 170.313]
  MoveL 180 to (190.33, 220.27, -6) mm, rotated rx -180 ry 0 rz 179.9 deg; joints [20.904, -39.586, 103.706, -156.826, 65.018, 170.321]
  MoveL 181 to (190.02, 220.36, -6) mm, rotated rx 180 ry 0 rz 179.9 deg; joints [20.905, -39.599, 103.736, -156.828, 65.034, 170.328]
  MoveL 182 to (189.72, 220.43, -6) mm, rotated rx 180 ry 0 rz 179.9 deg; joints [20.907, -39.611, 103.765, -156.829, 65.049, 170.334]
  MoveL 183 to (189.41, 220.49, -6) mm, rotated rx 180 ry 0 rz 179.9 deg; joints [20.909, -39.624, 103.793, -156.83, 65.064, 170.34]
  MoveL 184 to (189.1, 220.52, -6) mm, rotated rx 180 ry 0 rz 179.9 deg; joints [20.912, -39.636, 103.821, -156.829, 65.079, 170.345]
  MoveL 185 to (188.8, 220.53, -6) mm, rotated rx 180 ry 0 rz 179.9 deg; joints [20.916, -39.647, 103.848, -156.828, 65.094, 170.35]
  MoveL 186 to (187.57, 220.53, -6) mm, rotated rx 180 ry 0 rz 179.9 deg; joints [20.933, -39.694, 103.954, -156.821, 65.152, 170.369]
  MoveL 187 to (-186.96, 220.53, -6) mm, rotated rx 180 ry 0 rz 179.9 deg; joints [27.647, -51.185, 132.561, -152.021, 81.438, 176.178]
  MoveL 188 to (-187.26, 220.53, -6) mm, rotated rx -180 ry 0 rz 179.9 deg; joints [27.655, -51.192, 132.582, -152.015, 81.45, 176.184]
  MoveL 189 to (-187.57, 220.5, -6) mm, rotated rx 180 ry 0 rz 179.9 deg; joints [27.663, -51.199, 132.601, -152.007, 81.462, 176.189]
  MoveL 190 to (-187.88, 220.45, -6) mm, rotated rx -180 ry 0 rz 179.9 deg; joints [27.672, -51.205, 132.621, -151.999, 81.474, 176.193]
  MoveL 191 to (-188.18, 220.39, -6) mm, rotated rx 180 ry 0 rz 179.9 deg; joints [27.682, -51.212, 132.639, -151.99, 81.485, 176.198]
  MoveL 192 to (-188.49, 220.3, -6) mm, rotated rx 180 ry 0 rz 179.9 deg; joints [27.693, -51.218, 132.657, -151.979, 81.496, 176.202]
  MoveL 193 to (-188.8, 220.19, -6) mm, rotated rx 180 ry 0 rz 179.9 deg; joints [27.705, -51.224, 132.674, -151.968, 81.506, 176.205]
  MoveL 194 to (-189.1, 220.06, -6) mm, rotated rx 180 ry 0 rz 179.9 deg; joints [27.718, -51.23, 132.69, -151.956, 81.516, 176.208]
  MoveL 195 to (-189.41, 219.9, -6) mm, rotated rx -180 ry 0 rz 179.9 deg; joints [27.732, -51.236, 132.705, -151.942, 81.526, 176.211]
  MoveL 196 to (-189.72, 219.72, -6) mm, rotated rx 180 ry 0 rz 179.9 deg; joints [27.748, -51.241, 132.719, -151.927, 81.535, 176.214]
  MoveL 197 to (-190.02, 219.5, -6) mm, rotated rx -180 ry 0 rz 179.9 deg; joints [27.764, -51.245, 132.732, -151.911, 81.544, 176.215]
  MoveL 198 to (-190.31, 219.26, -6) mm, rotated rx -180 ry 0 rz 179.9 deg; joints [27.782, -51.249, 132.743, -151.894, 81.551, 176.216]
  MoveC 199 to (-191.1, 218.99, -6) mm, rotated rx 180 ry 0 rz 179.9 deg; joints [27.812, -51.265, 132.787, -151.865, 81.578, 176.226] to (-191.83, 219.41, -6) mm, rotated rx -180 ry 0 rz 179.9 deg; joints [27.81, -51.287, 132.852, -151.87, 81.615, 176.246]
  MoveL 200 to (-194.43, 223.17, -6) mm, rotated rx 180 ry 0 rz 179.9 deg; joints [27.705, -51.392, 133.163, -151.991, 81.79, 176.358]
  MoveC 201 to (-194.83, 223.75, -5.71) mm, rotated rx 180 ry 0 rz 179.9 deg; joints [27.688, -51.43, 133.214, -152.008, 81.8, 176.366] to (-195, 223.99, -5) mm, rotated rx 180 ry 0 rz 179.9 deg; joints [27.681, -51.491, 133.242, -152.013, 81.771, 176.351]
  Set speed (100.0 mm/s)
  MoveL 202 to (-195, 223.99, 6) mm, rotated rx 180 ry 0 rz 179.9 deg; joints [27.675, -52.328, 133.359, -151.968, 81.135, 176.011]
  MoveL 203 to (176.9, -186.06, 6) mm, rotated rx 180 ry 0 rz 179.9 deg; joints [34.188, -32.35, 85.948, -139.427, 59.739, 157.505]
  MoveL 204 to (176.9, -186.06, 1.5) mm, rotated rx 180 ry 0 rz 179.9 deg; joints [34.19, -32.137, 85.908, -139.491, 59.871, 157.634]
  Set speed (5.6 mm/s)
  MoveL 205 to (176.9, -186.06, -5) mm, rotated rx 180 ry 0 rz 179.9 deg; joints [34.193, -31.828, 85.848, -139.581, 60.062, 157.819]
  MoveC 206 to (177.13, -186.24, -5.71) mm, rotated rx 180 ry 0 rz 179.9 deg; joints [34.194, -31.779, 85.809, -139.584, 60.069, 157.826] to (177.68, -186.68, -6) mm, rotated rx 180 ry 0 rz 179.9 deg; joints [34.195, -31.729, 85.728, -139.57, 60.046, 157.801]
  Set speed (16.7 mm/s)
  MoveL 207 to (183.64, -191.36, -6) mm, rotated rx 180 ry 0 rz 179.9 deg; joints [34.213, -31.345, 84.889, -139.38, 59.707, 157.451]
  MoveL 208 to (183.72, -192.46, -6) mm, rotated rx 180 ry 0 rz 179.9 deg; joints [34.242, -31.31, 84.812, -139.333, 59.687, 157.403]
  MoveL 209 to (183.59, -192.6, -6) mm, rotated rx 180 ry 0 rz 179.9 deg; joints [34.249, -31.312, 84.815, -139.326, 59.69, 157.401]
  MoveL 210 to (-117.09, -192.6, -6) mm, rotated rx 180 ry 0 rz 179.9 deg; joints [41.002, -41.925, 108.435, -136.266, 71.597, 164.215]
  MoveL 211 to (-117.27, -192.46, -6) mm, rotated rx 180 ry 0 rz 179.9 deg; joints [41.002, -41.934, 108.455, -136.269, 71.605, 164.224]
  MoveL 212 to (-180.63, 207.46, -6) mm, rotated rx -180 ry 0 rz 179.9 deg; joints [28.073, -50.878, 131.659, -151.548, 80.945, 175.835]
  MoveL 213 to (-180.41, 207.64, -6) mm, rotated rx -180 ry 0 rz 179.9 deg; joints [28.06, -50.875, 131.651, -151.561, 80.939, 175.834]
  MoveL 214 to (183.59, 207.64, -6) mm, rotated rx -180 ry 0 rz 179.9 deg; joints [21.45, -39.661, 103.865, -156.249, 65.189, 170.117]
  MoveL 215 to (183.72, 207.46, -6) mm, rotated rx 180 ry 0 rz 179.9 deg; joints [21.455, -39.654, 103.848, -156.242, 65.181, 170.111]
  MoveL 216 to (183.72, -192.46, -6) mm, rotated rx 180 ry 0 rz 179.9 deg; joints [34.242, -31.31, 84.812, -139.333, 59.687, 157.403]
  Set speed (5.6 mm/s)
  MoveL 217 to (183.72, -192.46, -12) mm, rotated rx 180 ry 0 rz 179.9 deg; joints [34.245, -31.025, 84.752, -139.416, 59.859, 157.572]
  Set speed (16.7 mm/s)
  MoveL 218 to (183.59, -192.6, -12) mm, rotated rx 180 ry 0 rz 179.9 deg; joints [34.251, -31.027, 84.755, -139.409, 59.862, 157.57]
  MoveL 219 to (-117.09, -192.6, -12) mm, rotated rx -180 ry 0 rz 179.9 deg; joints [41.005, -41.586, 108.376, -136.327, 71.801, 164.419]
  MoveL 220 to (-117.27, -192.46, -12) mm, rotated rx 180 ry 0 rz 179.9 deg; joints [41.005, -41.595, 108.396, -136.33, 71.809, 164.427]
  MoveL 221 to (-180.22, 204.81, -12) mm, rotated rx 180 ry 0 rz 179.9 deg; joints [28.182, -50.39, 131.466, -151.461, 81.212, 175.962]
  MoveL 222 to (-180.43, 206.2, -12) mm, rotated rx 180 ry 0 rz 179.9 deg; joints [28.127, -50.411, 131.532, -151.519, 81.247, 175.991]
  MoveL 223 to (-180.22, 206.4, -12) mm, rotated rx 180 ry 0 rz 179.9 deg; joints [28.113, -50.408, 131.524, -151.533, 81.241, 175.99]
  MoveL 224 to (183.59, 206.4, -12) mm, rotated rx 180 ry 0 rz 179.9 deg; joints [21.496, -39.318, 103.765, -156.244, 65.42, 170.204]
  MoveL 225 to (183.72, 206.2, -12) mm, rotated rx 180 ry 0 rz 179.9 deg; joints [21.502, -39.31, 103.747, -156.236, 65.411, 170.197]
  MoveL 226 to (183.72, -192.46, -12) mm, rotated rx 180 ry 0 rz 179.9 deg; joints [34.245, -31.025, 84.752, -139.416, 59.859, 157.572]
  Set speed (5.6 mm/s)
  MoveL 227 to (183.72, -192.46, -18) mm, rotated rx -180 ry 0 rz 179.9 deg; joints [34.247, -30.738, 84.689, -139.497, 60.03, 157.739]
  Set speed (16.7 mm/s)
  MoveL 228 to (183.59, -192.6, -18) mm, rotated rx 180 ry 0 rz 179.9 deg; joints [34.254, -30.74, 84.692, -139.491, 60.033, 157.737]
  MoveL 229 to (-117.09, -192.6, -18) mm, rotated rx 180 ry 0 rz 179.9 deg; joints [41.008, -41.246, 108.315, -136.387, 72.003, 164.621]
  MoveL 230 to (-117.27, -192.46, -18) mm, rotated rx 180 ry 0 rz 179.9 deg; joints [41.009, -41.254, 108.335, -136.389, 72.012, 164.629]
  MoveL 231 to (-180.22, 204.81, -18) mm, rotated rx -180 ry 0 rz 179.9 deg; joints [28.185, -49.943, 131.395, -151.485, 81.542, 176.143]
  MoveL 232 to (-180.43, 206.2, -18) mm, rotated rx 180 ry 0 rz 179.9 deg; joints [28.13, -49.964, 131.46, -151.543, 81.577, 176.171]
  MoveL 233 to (-180.22, 206.4, -18) mm, rotated rx -180 ry 0 rz 179.9 deg; joints [28.116, -49.961, 131.453, -151.557, 81.572, 176.171]
  MoveL 234 to (183.59, 206.4, -18) mm, rotated rx -180 ry 0 rz 179.9 deg; joints [21.499, -38.991, 103.704, -156.29, 65.663, 170.321]
  MoveL 235 to (183.72, 206.2, -18) mm, rotated rx -180 ry 0 rz 179.9 deg; joints [21.504, -38.983, 103.685, -156.282, 65.655, 170.314]
  MoveL 236 to (183.72, -192.46, -18) mm, rotated rx -180 ry 0 rz 179.9 deg; joints [34.247, -30.738, 84.689, -139.497, 60.03, 157.739]
  Set speed (5.6 mm/s)
  MoveL 237 to (183.72, -192.46, -20.05) mm, rotated rx 180 ry 0 rz 179.9 deg; joints [34.248, -30.64, 84.667, -139.525, 60.088, 157.795]
  Set speed (16.7 mm/s)
  MoveL 238 to (183.59, -192.6, -20.05) mm, rotated rx -180 ry 0 rz 179.9 deg; joints [34.254, -30.641, 84.67, -139.518, 60.092, 157.793]
  MoveL 239 to (-117.09, -192.6, -20.05) mm, rotated rx 180 ry 0 rz 179.9 deg; joints [41.009, -41.129, 108.294, -136.407, 72.072, 164.689]
  MoveL 240 to (-117.27, -192.46, -20.05) mm, rotated rx 180 ry 0 rz 179.9 deg; joints [41.01, -41.138, 108.314, -136.409, 72.081, 164.697]
  MoveL 241 to (-180.22, 204.81, -20.05) mm, rotated rx -180 ry 0 rz 179.9 deg; joints [28.186, -49.79, 131.37, -151.492, 81.655, 176.204]
  MoveL 242 to (-180.43, 206.2, -20.05) mm, rotated rx 180 ry 0 rz 179.9 deg; joints [28.131, -49.811, 131.435, -151.551, 81.69, 176.233]
  MoveL 243 to (-180.22, 206.4, -20.05) mm, rotated rx 180 ry 0 rz 179.9 deg; joints [28.117, -49.808, 131.427, -151.565, 81.684, 176.232]
  MoveL 244 to (183.59, 206.4, -20.05) mm, rotated rx 180 ry 0 rz 179.9 deg; joints [21.499, -38.879, 103.682, -156.306, 65.746, 170.36]
  MoveL 245 to (183.72, 206.2, -20.05) mm, rotated rx 180 ry 0 rz 179.9 deg; joints [21.505, -38.871, 103.664, -156.298, 65.737, 170.354]
  MoveL 246 to (183.72, -192.46, -20.05) mm, rotated rx 180 ry 0 rz 179.9 deg; joints [34.248, -30.64, 84.667, -139.525, 60.088, 157.795]
  Set speed (100.0 mm/s)
  MoveL 247 to (183.72, -192.46, 6) mm, rotated rx -180 ry 0 rz 179.9 deg; joints [34.237, -31.878, 84.923, -139.163, 59.339, 157.06]
  MoveL 248 to (-122.54, -205.85, 6) mm, rotated rx 180 ry 0 rz 179.9 deg; joints [41.532, -42.429, 108.125, -135.539, 71.162, 163.455]
  MoveL 249 to (-122.54, -205.85, 5.17) mm, rotated rx -180 ry 0 rz 179.9 deg; joints [41.533, -42.383, 108.118, -135.548, 71.19, 163.484]
  Set speed (5.6 mm/s)
  MoveL 250 to (-122.54, -205.85, -4.96) mm, rotated rx 180 ry 0 rz 179.9 deg; joints [41.538, -41.815, 108.028, -135.655, 71.533, 163.835]
  Set speed (16.7 mm/s)
  MoveL 251 to (-122.46, -205.97, -5.48) mm, rotated rx -180 ry 0 rz 179.9 deg; joints [41.54, -41.781, 108.011, -135.657, 71.546, 163.847]
  MoveL 252 to (-122.4, -206.34, -5.86) mm, rotated rx 180 ry 0 rz 179.9 deg; joints [41.55, -41.748, 107.981, -135.648, 71.55, 163.846]
  MoveL 253 to (-122.65, -206.78, -6) mm, rotated rx -180 ry 0 rz 179.9 deg; joints [41.569, -41.737, 107.97, -135.628, 71.556, 163.841]
  MoveL 254 to (-123.23, -207.24, -6) mm, rotated rx 180 ry 0 rz 179.9 deg; joints [41.598, -41.742, 107.982, -135.6, 71.569, 163.836]
  MoveL 255 to (-123.55, -207.56, -6) mm, rotated rx 180 ry 0 rz 179.9 deg; joints [41.616, -41.744, 107.984, -135.582, 71.575, 163.832]
  MoveL 256 to (-123.82, -207.88, -6) mm, rotated rx 180 ry 0 rz 179.9 deg; joints [41.633, -41.744, 107.983, -135.565, 71.579, 163.826]
  MoveL 257 to (-124.09, -208.26, -6) mm, rotated rx -180 ry 0 rz 179.9 deg; joints [41.651, -41.742, 107.978, -135.546, 71.582, 163.818]
  MoveL 258 to (-124.31, -208.65, -6) mm, rotated rx 180 ry 0 rz 179.9 deg; joints [41.668, -41.739, 107.97, -135.527, 71.583, 163.809]
  MoveL 259 to (-124.46, -208.96, -6) mm, rotated rx 180 ry 0 rz 179.9 deg; joints [41.681, -41.735, 107.961, -135.513, 71.583, 163.801]
  MoveL 260 to (-124.58, -209.27, -6) mm, rotated rx 180 ry 0 rz 179.9 deg; joints [41.694, -41.731, 107.951, -135.499, 71.582, 163.793]
  MoveL 261 to (-124.67, -209.57, -6) mm, rotated rx -180 ry 0 rz 179.9 deg; joints [41.705, -41.726, 107.939, -135.486, 71.58, 163.785]
  MoveL 262 to (-124.75, -209.88, -6) mm, rotated rx 180 ry 0 rz 179.9 deg; joints [41.716, -41.721, 107.926, -135.473, 71.578, 163.776]
  MoveL 263 to (-124.78, -210.03, -6) mm, rotated rx 180 ry 0 rz 179.9 deg; joints [41.722, -41.718, 107.919, -135.467, 71.576, 163.771]
  MoveL 264 to (-124.81, -210.19, -6) mm, rotated rx -180 ry 0 rz 179.9 deg; joints [41.727, -41.715, 107.911, -135.46, 71.575, 163.766]
  MoveL 265 to (-124.83, -210.34, -6) mm, rotated rx 180 ry 0 rz 179.9 deg; joints [41.732, -41.711, 107.904, -135.454, 71.573, 163.761]
  MoveL 266 to (-124.84, -210.49, -6) mm, rotated rx 180 ry 0 rz 179.9 deg; joints [41.737, -41.708, 107.895, -135.448, 71.571, 163.756]
  MoveL 267 to (-124.85, -210.65, -6) mm, rotated rx -180 ry 0 rz 179.9 deg; joints [41.742, -41.704, 107.887, -135.442, 71.569, 163.751]
  MoveL 268 to (-124.86, -210.8, -6) mm, rotated rx 180 ry 0 rz 179.9 deg; joints [41.746, -41.701, 107.878, -135.436, 71.566, 163.746]
  MoveL 269 to (-124.86, -210.95, -6) mm, rotated rx 180 ry 0 rz 179.9 deg; joints [41.751, -41.697, 107.869, -135.43, 71.564, 163.741]
  MoveL 270 to (-124.86, -211.11, -6) mm, rotated rx -180 ry 0 rz 179.9 deg; joints [41.755, -41.693, 107.86, -135.425, 71.561, 163.735]
  MoveL 271 to (-124.85, -211.26, -6) mm, rotated rx -180 ry 0 rz 179.9 deg; joints [41.76, -41.689, 107.85, -135.419, 71.559, 163.73]
  MoveL 272 to (-124.84, -211.41, -6) mm, rotated rx 180 ry 0 rz 179.9 deg; joints [41.764, -41.685, 107.84, -135.413, 71.556, 163.724]
  MoveL 273 to (-124.82, -211.57, -6) mm, rotated rx 180 ry 0 rz 179.9 deg; joints [41.768, -41.68, 107.83, -135.408, 71.553, 163.718]
  MoveL 274 to (-124.8, -211.72, -6) mm, rotated rx 180 ry 0 rz 179.9 deg; joints [41.772, -41.676, 107.819, -135.402, 71.549, 163.713]
  MoveL 275 to (-124.7, -212.33, -6) mm, rotated rx 180 ry 0 rz 179.9 deg; joints [41.787, -41.658, 107.776, -135.381, 71.536, 163.689]
  MoveL 276 to (-124.64, -212.64, -6) mm, rotated rx 180 ry 0 rz 179.9 deg; joints [41.795, -41.648, 107.753, -135.37, 71.529, 163.678]
  MoveL 277 to (-124.56, -212.95, -6) mm, rotated rx 180 ry 0 rz 179.9 deg; joints [41.802, -41.638, 107.729, -135.36, 71.521, 163.665]
  MoveL 278 to (-124.45, -213.25, -6) mm, rotated rx -180 ry 0 rz 179.9 deg; joints [41.808, -41.627, 107.704, -135.35, 71.512, 163.653]
  MoveL 279 to (-124.33, -213.56, -6) mm, rotated rx 180 ry 0 rz 179.9 deg; joints [41.814, -41.616, 107.677, -135.341, 71.503, 163.639]
  MoveL 280 to (-124.22, -213.78, -6) mm, rotated rx 180 ry 0 rz 179.9 deg; joints [41.817, -41.607, 107.657, -135.335, 71.496, 163.63]
  MoveL 281 to (-124.1, -214, -6) mm, rotated rx -180 ry 0 rz 179.9 deg; joints [41.82, -41.598, 107.636, -135.328, 71.488, 163.62]
  MoveL 282 to (-123.97, -214.22, -6) mm, rotated rx 180 ry 0 rz 179.9 deg; joints [41.823, -41.589, 107.614, -135.322, 71.48, 163.609]
  MoveL 283 to (-123.82, -214.43, -6) mm, rotated rx 180 ry 0 rz 179.9 deg; joints [41.826, -41.579, 107.591, -135.317, 71.471, 163.599]
  MoveL 284 to (-123.63, -214.68, -6) mm, rotated rx -180 ry 0 rz 179.9 deg; joints [41.828, -41.567, 107.563, -135.311, 71.46, 163.586]
  MoveL 285 to (-123.41, -214.93, -6) mm, rotated rx -180 ry 0 rz 179.9 deg; joints [41.83, -41.555, 107.534, -135.305, 71.449, 163.573]
  MoveL 286 to (-123.14, -215.19, -6) mm, rotated rx 180 ry 0 rz 179.9 deg; joints [41.83, -41.54, 107.499, -135.3, 71.435, 163.559]
  MoveL 287 to (-122.87, -215.42, -6) mm, rotated rx -180 ry 0 rz 179.9 deg; joints [41.83, -41.526, 107.468, -135.296, 71.422, 163.545]
  MoveL 288 to (-122.64, -215.6, -6) mm, rotated rx 180 ry 0 rz 179.9 deg; joints [41.829, -41.515, 107.441, -135.294, 71.411, 163.534]
  MoveL 289 to (-122.4, -215.76, -6) mm, rotated rx 180 ry 0 rz 179.9 deg; joints [41.827, -41.504, 107.416, -135.292, 71.4, 163.524]
  MoveL 290 to (-122.16, -215.89, -6) mm, rotated rx -180 ry 0 rz 179.9 deg; joints [41.825, -41.494, 107.391, -135.291, 71.39, 163.515]
  MoveL 291 to (-121.92, -216.02, -6) mm, rotated rx 180 ry 0 rz 179.9 deg; joints [41.822, -41.484, 107.368, -135.29, 71.38, 163.506]
  MoveL 292 to (-121.65, -216.14, -6) mm, rotated rx 180 ry 0 rz 179.9 deg; joints [41.819, -41.472, 107.342, -135.291, 71.368, 163.496]
  MoveL 293 to (-121.37, -216.24, -6) mm, rotated rx -180 ry 0 rz 179.9 deg; joints [41.814, -41.462, 107.317, -135.292, 71.357, 163.487]
  MoveL 294 to (-121.06, -216.33, -6) mm, rotated rx -180 ry 0 rz 179.9 deg; joints [41.809, -41.45, 107.291, -135.293, 71.345, 163.477]
  MoveL 295 to (-120.76, -216.41, -6) mm, rotated rx -180 ry 0 rz 179.9 deg; joints [41.803, -41.44, 107.266, -135.296, 71.333, 163.469]
  MoveL 296 to (-120.45, -216.46, -6) mm, rotated rx 180 ry 0 rz 179.9 deg; joints [41.796, -41.429, 107.243, -135.3, 71.322, 163.461]
  MoveL 297 to (-120.14, -216.49, -6) mm, rotated rx 180 ry 0 rz 179.9 deg; joints [41.789, -41.419, 107.22, -135.304, 71.31, 163.453]
  MoveL 298 to (-118.92, -216.5, -6) mm, rotated rx -180 ry 0 rz 179.9 deg; joints [41.758, -41.383, 107.136, -135.325, 71.268, 163.428]
  MoveL 299 to (182.67, -216.5, -6) mm, rotated rx 180 ry 0 rz 179.9 deg; joints [34.934, -30.659, 83.37, -138.289, 59.365, 156.437]
  MoveL 300 to (188.8, -216.5, -6) mm, rotated rx -180 ry 0 rz 179.9 deg; joints [34.815, -30.394, 82.797, -138.294, 59.088, 156.261]
  MoveL 301 to (189.1, -216.49, -6) mm, rotated rx 180 ry 0 rz 179.9 deg; joints [34.809, -30.381, 82.769, -138.294, 59.074, 156.253]
  MoveL 302 to (189.41, -216.46, -6) mm, rotated rx 180 ry 0 rz 179.9 deg; joints [34.802, -30.368, 82.743, -138.296, 59.061, 156.246]
  MoveL 303 to (189.72, -216.4, -6) mm, rotated rx 180 ry 0 rz 179.9 deg; joints [34.795, -30.357, 82.717, -138.298, 59.048, 156.239]
  MoveL 304 to (190.02, -216.33, -6) mm, rotated rx 180 ry 0 rz 179.9 deg; joints [34.787, -30.345, 82.693, -138.302, 59.035, 156.233]
  MoveL 305 to (190.45, -216.2, -6) mm, rotated rx 180 ry 0 rz 179.9 deg; joints [34.775, -30.331, 82.662, -138.308, 59.017, 156.227]
  MoveL 306 to (190.87, -216.02, -6) mm, rotated rx 180 ry 0 rz 179.9 deg; joints [34.762, -30.318, 82.634, -138.316, 59.001, 156.222]
  MoveL 307 to (191.27, -215.8, -6) mm, rotated rx -180 ry 0 rz 179.9 deg; joints [34.748, -30.307, 82.61, -138.325, 58.986, 156.22]
  MoveL 308 to (191.47, -215.68, -6) mm, rotated rx -180 ry 0 rz 179.9 deg; joints [34.741, -30.301, 82.6, -138.331, 58.979, 156.219]
  MoveL 309 to (191.67, -215.54, -6) mm, rotated rx -180 ry 0 rz 179.9 deg; joints [34.733, -30.297, 82.59, -138.337, 58.972, 156.219]
  MoveL 310 to (191.87, -215.38, -6) mm, rotated rx 180 ry 0 rz 179.9 deg; joints [34.725, -30.293, 82.581, -138.344, 58.965, 156.22]
  MoveL 311 to (192.08, -215.21, -6) mm, rotated rx -180 ry 0 rz 179.9 deg; joints [34.716, -30.289, 82.573, -138.351, 58.959, 156.222]
  MoveL 312 to (192.29, -215.01, -6) mm, rotated rx 180 ry 0 rz 179.9 deg; joints [34.707, -30.286, 82.567, -138.36, 58.952, 156.224]
  MoveL 313 to (192.48, -214.81, -6) mm, rotated rx 180 ry 0 rz 179.9 deg; joints [34.698, -30.284, 82.562, -138.369, 58.947, 156.227]
  MoveL 314 to (192.73, -214.49, -6) mm, rotated rx 180 ry 0 rz 179.9 deg; joints [34.684, -30.282, 82.559, -138.383, 58.94, 156.233]
  MoveL 315 to (192.94, -214.18, -6) mm, rotated rx 180 ry 0 rz 179.9 deg; joints [34.671, -30.282, 82.559, -138.397, 58.935, 156.24]
  MoveL 316 to (193.12, -213.87, -6) mm, rotated rx 180 ry 0 rz 179.9 deg; joints [34.659, -30.283, 82.562, -138.41, 58.931, 156.248]
  MoveL 317 to (193.28, -213.56, -6) mm, rotated rx -180 ry 0 rz 179.9 deg; joints [34.648, -30.285, 82.568, -138.424, 58.929, 156.257]
  MoveL 318 to (193.4, -213.25, -6) mm, rotated rx 180 ry 0 rz 179.9 deg; joints [34.637, -30.289, 82.576, -138.438, 58.928, 156.266]
  MoveL 319 to (193.51, -212.95, -6) mm, rotated rx 180 ry 0 rz 179.9 deg; joints [34.626, -30.294, 82.586, -138.451, 58.928, 156.276]
  MoveL 320 to (193.59, -212.64, -6) mm, rotated rx -180 ry 0 rz 179.9 deg; joints [34.616, -30.299, 82.598, -138.464, 58.929, 156.287]
  MoveL 321 to (193.65, -212.33, -6) mm, rotated rx 180 ry 0 rz 179.9 deg; joints [34.607, -30.305, 82.613, -138.478, 58.931, 156.298]
  MoveL 322 to (193.69, -212.03, -6) mm, rotated rx 180 ry 0 rz 179.9 deg; joints [34.597, -30.313, 82.629, -138.491, 58.934, 156.31]
  MoveL 323 to (193.72, -211.72, -6) mm, rotated rx -180 ry 0 rz 179.9 deg; joints [34.588, -30.321, 82.646, -138.505, 58.938, 156.322]
  MoveL 324 to (193.72, -211.11, -6) mm, rotated rx 180 ry 0 rz 179.9 deg; joints [34.571, -30.339, 82.686, -138.532, 58.947, 156.348]
  MoveL 325 to (193.72, -210.8, -6) mm, rotated rx -180 ry 0 rz 179.9 deg; joints [34.563, -30.348, 82.706, -138.545, 58.952, 156.361]
  MoveL 326 to (193.71, -210.65, -6) mm, rotated rx 180 ry 0 rz 179.9 deg; joints [34.559, -30.353, 82.717, -138.552, 58.954, 156.368]
  MoveL 327 to (193.7, -210.49, -6) mm, rotated rx -180 ry 0 rz 179.9 deg; joints [34.555, -30.358, 82.728, -138.558, 58.957, 156.374]
  MoveL 328 to (193.69, -210.34, -6) mm, rotated rx -180 ry 0 rz 179.9 deg; joints [34.551, -30.363, 82.739, -138.565, 58.96, 156.381]
  MoveL 329 to (193.67, -210.19, -6) mm, rotated rx 180 ry 0 rz 179.9 deg; joints [34.547, -30.368, 82.751, -138.572, 58.963, 156.388]
  MoveL 330 to (193.64, -210.03, -6) mm, rotated rx 180 ry 0 rz 179.9 deg; joints [34.543, -30.374, 82.763, -138.579, 58.967, 156.396]
  MoveL 331 to (193.61, -209.88, -6) mm, rotated rx 180 ry 0 rz 179.9 deg; joints [34.539, -30.38, 82.776, -138.585, 58.971, 156.403]
  MoveL 332 to (193.57, -209.73, -6) mm, rotated rx -180 ry 0 rz 179.9 deg; joints [34.536, -30.386, 82.79, -138.592, 58.975, 156.41]
  MoveL 333 to (193.53, -209.57, -6) mm, rotated rx 180 ry 0 rz 179.9 deg; joints [34.532, -30.392, 82.803, -138.599, 58.979, 156.418]
  MoveL 334 to (193.49, -209.42, -6) mm, rotated rx 180 ry 0 rz 179.9 deg; joints [34.529, -30.399, 82.818, -138.605, 58.983, 156.426]
  MoveL 335 to (193.44, -209.27, -6) mm, rotated rx -180 ry 0 rz 179.9 deg; joints [34.526, -30.405, 82.832, -138.612, 58.988, 156.434]
  MoveL 336 to (193.38, -209.11, -6) mm, rotated rx -180 ry 0 rz 179.9 deg; joints [34.522, -30.412, 82.848, -138.619, 58.993, 156.442]
  MoveL 337 to (193.32, -208.96, -6) mm, rotated rx -180 ry 0 rz 179.9 deg; joints [34.519, -30.42, 82.864, -138.625, 58.998, 156.45]
  MoveL 338 to (193.25, -208.8, -6) mm, rotated rx 180 ry 0 rz 179.9 deg; joints [34.516, -30.427, 82.88, -138.632, 59.004, 156.459]
  MoveL 339 to (193.17, -208.65, -6) mm, rotated rx 180 ry 0 rz 179.9 deg; joints [34.514, -30.435, 82.897, -138.639, 59.01, 156.467]
  MoveL 340 to (193.03, -208.4, -6) mm, rotated rx 180 ry 0 rz 179.9 deg; joints [34.509, -30.449, 82.927, -138.65, 59.02, 156.482]
  MoveL 341 to (192.87, -208.14, -6) mm, rotated rx -180 ry 0 rz 179.9 deg; joints [34.505, -30.463, 82.959, -138.661, 59.031, 156.497]
  MoveL 342 to (192.69, -207.88, -6) mm, rotated rx -180 ry 0 rz 179.9 deg; joints [34.502, -30.479, 82.993, -138.672, 59.044, 156.514]
  MoveL 343 to (192.48, -207.63, -6) mm, rotated rx 180 ry 0 rz 179.9 deg; joints [34.498, -30.495, 83.029, -138.683, 59.057, 156.53]
  MoveL 344 to (192.21, -207.35, -6) mm, rotated rx 180 ry 0 rz 179.9 deg; joints [34.496, -30.515, 83.072, -138.695, 59.074, 156.55]
  MoveL 345 to (191.94, -207.1, -6) mm, rotated rx 180 ry 0 rz 179.9 deg; joints [34.494, -30.534, 83.113, -138.706, 59.09, 156.568]
  MoveL 346 to (191.67, -206.89, -6) mm, rotated rx -180 ry 0 rz 179.9 deg; joints [34.493, -30.552, 83.152, -138.715, 59.105, 156.584]
  MoveL 347 to (191.4, -206.71, -6) mm, rotated rx 180 ry 0 rz 179.9 deg; joints [34.493, -30.569, 83.189, -138.723, 59.12, 156.599]
  MoveL 348 to (190.87, -206.41, -6) mm, rotated rx 180 ry 0 rz 179.9 deg; joints [34.496, -30.601, 83.258, -138.735, 59.149, 156.627]
  MoveL 349 to (190.33, -206.2, -6) mm, rotated rx -180 ry 0 rz 179.9 deg; joints [34.5, -30.63, 83.322, -138.744, 59.177, 156.651]
  MoveL 350 to (190.26, -206.17, -6) mm, rotated rx 180 ry 0 rz 179.9 deg; joints [34.501, -30.634, 83.331, -138.745, 59.181, 156.655]
  MoveL 351 to (190.02, -206.1, -6) mm, rotated rx 180 ry 0 rz 179.9 deg; joints [34.503, -30.647, 83.357, -138.748, 59.192, 156.664]
  MoveL 352 to (189.72, -206.03, -6) mm, rotated rx -180 ry 0 rz 179.9 deg; joints [34.507, -30.662, 83.391, -138.751, 59.207, 156.676]
  MoveL 353 to (189.41, -205.98, -6) mm, rotated rx 180 ry 0 rz 179.9 deg; joints [34.511, -30.677, 83.423, -138.753, 59.222, 156.687]
  MoveL 354 to (189.1, -205.94, -6) mm, rotated rx -180 ry 0 rz 179.9 deg; joints [34.516, -30.691, 83.453, -138.754, 59.236, 156.697]
  MoveL 355 to (188.8, -205.93, -6) mm, rotated rx -180 ry 0 rz 179.9 deg; joints [34.522, -30.705, 83.483, -138.755, 59.251, 156.706]
  MoveL 356 to (187.57, -205.93, -6) mm, rotated rx -180 ry 0 rz 179.9 deg; joints [34.545, -30.758, 83.598, -138.754, 59.306, 156.741]
  MoveL 357 to (-118.92, -205.93, -6) mm, rotated rx -180 ry 0 rz 179.9 deg; joints [41.446, -41.649, 107.77, -135.726, 71.441, 163.795]
  MoveL 358 to (-120.14, -205.94, -6) mm, rotated rx 180 ry 0 rz 179.9 deg; joints [41.479, -41.685, 107.852, -135.704, 71.483, 163.82]
  MoveL 359 to (-120.76, -206.01, -6) mm, rotated rx 180 ry 0 rz 179.9 deg; joints [41.497, -41.701, 107.889, -135.691, 71.503, 163.829]
  MoveL 360 to (-121.37, -206.16, -6) mm, rotated rx -180 ry 0 rz 179.9 deg; joints [41.517, -41.715, 107.921, -135.674, 71.522, 163.836]
  MoveL 361 to (-121.47, -206.2, -6) mm, rotated rx -180 ry 0 rz 179.9 deg; joints [41.521, -41.717, 107.926, -135.671, 71.525, 163.837]
  MoveL 362 to (-122.06, -206.44, -6) mm, rotated rx -180 ry 0 rz 179.9 deg; joints [41.544, -41.728, 107.951, -135.651, 71.541, 163.841]
  MoveL 363 to (-122.65, -206.78, -6) mm, rotated rx -180 ry 0 rz 179.9 deg; joints [41.569, -41.737, 107.97, -135.628, 71.556, 163.841]
  MoveC 364 to (-123.38, -206.98, -6) mm, rotated rx 180 ry 0 rz 179.9 deg; joints [41.595, -41.753, 108.007, -135.607, 71.578, 163.848] to (-124.05, -206.61, -6) mm, rotated rx 180 ry 0 rz 179.9 deg; joints [41.601, -41.782, 108.074, -135.609, 71.607, 163.875]
  MoveL 365 to (-124.96, -206.23, -6) mm, rotated rx -180 ry 0 rz 179.9 deg; joints [41.614, -41.818, 108.158, -135.607, 71.645, 163.906]
  MoveL 366 to (-128.18, -206.64, -6) mm, rotated rx -180 ry 0 rz 179.9 deg; joints [41.711, -41.901, 108.349, -135.534, 71.749, 163.956]
  Set speed (5.6 mm/s)
  MoveL 367 to (-128.18, -206.64, -11) mm, rotated rx -180 ry 0 rz 179.9 deg; joints [41.714, -41.619, 108.3, -135.585, 71.917, 164.127]
  MoveC 368 to (-127.89, -206.6, -11.71) mm, rotated rx 180 ry 0 rz 179.9 deg; joints [41.705, -41.572, 108.277, -135.599, 71.931, 164.147] to (-127.19, -206.49, -12) mm, rotated rx -180 ry 0 rz 179.9 deg; joints [41.684, -41.538, 108.234, -135.619, 71.919, 164.147]
  Set speed (16.7 mm/s)
  MoveC 369 to (-126.45, -206.66, -12) mm, rotated rx 180 ry 0 rz 179.9 deg; joints [41.669, -41.512, 108.173, -135.626, 71.89, 164.126] to (-126.05, -207.32, -12) mm, rotated rx 180 ry 0 rz 179.9 deg; joints [41.678, -41.484, 108.108, -135.608, 71.866, 164.095]
  MoveL 370 to (-125.06, -213.56, -12) mm, rotated rx 180 ry 0 rz 179.9 deg; joints [41.836, -41.3, 107.668, -135.39, 71.727, 163.859]
  MoveL 371 to (-124.66, -216.02, -12) mm, rotated rx 180 ry 0 rz 179.9 deg; joints [41.898, -41.227, 107.494, -135.304, 71.673, 163.766]
  MoveL 372 to (-124.61, -216.25, -12) mm, rotated rx 180 ry 0 rz 179.9 deg; joints [41.903, -41.22, 107.476, -135.296, 71.667, 163.757]
  MoveL 373 to (-124.54, -216.49, -12) mm, rotated rx 180 ry 0 rz 179.9 deg; joints [41.908, -41.212, 107.457, -135.288, 71.661, 163.747]
  MoveL 374 to (-124.46, -216.73, -12) mm, rotated rx 180 ry 0 rz 179.9 deg; joints [41.913, -41.204, 107.437, -135.281, 71.654, 163.737]
  MoveL 375 to (-124.36, -216.96, -12) mm, rotated rx 180 ry 0 rz 179.9 deg; joints [41.917, -41.195, 107.417, -135.274, 71.647, 163.727]
  MoveL 376 to (-124.25, -217.2, -12) mm, rotated rx 180 ry 0 rz 179.9 deg; joints [41.921, -41.186, 107.395, -135.267, 71.639, 163.716]
  MoveL 377 to (-124.12, -217.44, -12) mm, rotated rx -180 ry 0 rz 179.9 deg; joints [41.925, -41.176, 107.372, -135.26, 71.631, 163.706]
  MoveL 378 to (-123.98, -217.67, -12) mm, rotated rx -180 ry 0 rz 179.9 deg; joints [41.928, -41.166, 107.349, -135.253, 71.622, 163.694]
  MoveL 379 to (-123.82, -217.91, -12) mm, rotated rx 180 ry 0 rz 179.9 deg; joints [41.931, -41.155, 107.324, -135.247, 71.612, 163.683]
  MoveL 380 to (-123.6, -218.19, -12) mm, rotated rx 180 ry 0 rz 179.9 deg; joints [41.933, -41.142, 107.292, -135.241, 71.6, 163.669]
  MoveL 381 to (-123.35, -218.47, -12) mm, rotated rx 180 ry 0 rz 179.9 deg; joints [41.935, -41.128, 107.258, -135.235, 71.587, 163.654]
  MoveL 382 to (-123.1, -218.71, -12) mm, rotated rx -180 ry 0 rz 179.9 deg; joints [41.935, -41.114, 107.227, -135.23, 71.574, 163.641]
  MoveL 383 to (-122.85, -218.91, -12) mm, rotated rx 180 ry 0 rz 179.9 deg; joints [41.935, -41.102, 107.198, -135.226, 71.562, 163.628]
  MoveL 384 to (-122.61, -219.1, -12) mm, rotated rx -180 ry 0 rz 179.9 deg; joints [41.934, -41.09, 107.17, -135.224, 71.551, 163.617]
  MoveL 385 to (-122.36, -219.26, -12) mm, rotated rx 180 ry 0 rz 179.9 deg; joints [41.932, -41.079, 107.144, -135.222, 71.539, 163.606]
  MoveL 386 to (-122.11, -219.4, -12) mm, rotated rx 180 ry 0 rz 179.9 deg; joints [41.929, -41.068, 107.119, -135.221, 71.528, 163.596]
  MoveL 387 to (-121.86, -219.52, -12) mm, rotated rx -180 ry 0 rz 179.9 deg; joints [41.926, -41.058, 107.095, -135.221, 71.518, 163.587]
  MoveL 388 to (-121.62, -219.63, -12) mm, rotated rx 180 ry 0 rz 179.9 deg; joints [41.923, -41.048, 107.072, -135.221, 71.508, 163.578]
  MoveL 389 to (-121.37, -219.72, -12) mm, rotated rx 180 ry 0 rz 179.9 deg; joints [41.919, -41.039, 107.05, -135.222, 71.498, 163.57]
  MoveL 390 to (-121.06, -219.81, -12) mm, rotated rx -180 ry 0 rz 179.9 deg; joints [41.914, -41.027, 107.024, -135.224, 71.485, 163.561]
  MoveL 391 to (-120.76, -219.88, -12) mm, rotated rx -180 ry 0 rz 179.9 deg; joints [41.908, -41.017, 106.999, -135.227, 71.474, 163.552]
  MoveL 392 to (-120.45, -219.93, -12) mm, rotated rx -180 ry 0 rz 179.9 deg; joints [41.901, -41.006, 106.975, -135.23, 71.462, 163.544]
  MoveL 393 to (-120.14, -219.97, -12) mm, rotated rx 180 ry 0 rz 179.9 deg; joints [41.894, -40.997, 106.952, -135.235, 71.451, 163.536]
  MoveL 394 to (-118.92, -219.98, -12) mm, rotated rx -180 ry 0 rz 179.9 deg; joints [41.862, -40.96, 106.869, -135.255, 71.408, 163.511]
  MoveL 395 to (182.67, -219.98, -12) mm, rotated rx 180 ry 0 rz 179.9 deg; joints [35.033, -30.273, 83.083, -138.223, 59.479, 156.461]
  MoveL 396 to (188.8, -219.98, -12) mm, rotated rx 180 ry 0 rz 179.9 deg; joints [34.914, -30.008, 82.509, -138.227, 59.2, 156.285]
  MoveL 397 to (189.1, -219.96, -12) mm, rotated rx -180 ry 0 rz 179.9 deg; joints [34.908, -29.995, 82.481, -138.228, 59.187, 156.276]
  MoveL 398 to (189.41, -219.93, -12) mm, rotated rx -180 ry 0 rz 179.9 deg; joints [34.901, -29.983, 82.454, -138.23, 59.173, 156.269]
  MoveL 399 to (189.72, -219.88, -12) mm, rotated rx 180 ry 0 rz 179.9 deg; joints [34.893, -29.971, 82.429, -138.232, 59.16, 156.262]
  MoveL 400 to (190.02, -219.81, -12) mm, rotated rx 180 ry 0 rz 179.9 deg; joints [34.885, -29.96, 82.405, -138.236, 59.147, 156.256]
  MoveL 401 to (190.31, -219.72, -12) mm, rotated rx 180 ry 0 rz 179.9 deg; joints [34.878, -29.95, 82.384, -138.239, 59.136, 156.252]
  MoveL 402 to (190.59, -219.62, -12) mm, rotated rx -180 ry 0 rz 179.9 deg; joints [34.869, -29.941, 82.364, -138.244, 59.124, 156.248]
  MoveL 403 to (190.88, -219.49, -12) mm, rotated rx -180 ry 0 rz 179.9 deg; joints [34.86, -29.932, 82.345, -138.25, 59.113, 156.245]
  MoveL 404 to (191.16, -219.34, -12) mm, rotated rx 180 ry 0 rz 179.9 deg; joints [34.851, -29.924, 82.328, -138.256, 59.102, 156.243]
  MoveL 405 to (191.45, -219.17, -12) mm, rotated rx -180 ry 0 rz 179.9 deg; joints [34.84, -29.917, 82.312, -138.264, 59.092, 156.242]
  MoveL 406 to (191.73, -218.97, -12) mm, rotated rx 180 ry 0 rz 179.9 deg; joints [34.829, -29.91, 82.299, -138.273, 59.082, 156.242]
  MoveL 407 to (192.02, -218.74, -12) mm, rotated rx 180 ry 0 rz 179.9 deg; joints [34.818, -29.905, 82.287, -138.283, 59.073, 156.244]
  MoveL 408 to (192.3, -218.47, -12) mm, rotated rx -180 ry 0 rz 179.9 deg; joints [34.805, -29.9, 82.278, -138.295, 59.064, 156.247]
  MoveL 409 to (192.48, -218.28, -12) mm, rotated rx 180 ry 0 rz 179.9 deg; joints [34.796, -29.898, 82.274, -138.303, 59.059, 156.25]
  MoveL 410 to (192.71, -218, -12) mm, rotated rx 180 ry 0 rz 179.9 deg; joints [34.784, -29.897, 82.271, -138.315, 59.053, 156.255]
  MoveL 411 to (192.91, -217.71, -12) mm, rotated rx -180 ry 0 rz 179.9 deg; joints [34.772, -29.896, 82.27, -138.328, 59.048, 156.261]
  MoveL 412 to (193.08, -217.43, -12) mm, rotated rx 180 ry 0 rz 179.9 deg; joints [34.761, -29.897, 82.273, -138.34, 59.045, 156.268]
  MoveL 413 to (193.23, -217.15, -12) mm, rotated rx -180 ry 0 rz 179.9 deg; joints [34.75, -29.899, 82.277, -138.353, 59.042, 156.276]
  MoveL 414 to (193.35, -216.87, -12) mm, rotated rx 180 ry 0 rz 179.9 deg; joints [34.74, -29.902, 82.284, -138.365, 59.041, 156.285]
  MoveL 415 to (193.46, -216.58, -12) mm, rotated rx -180 ry 0 rz 179.9 deg; joints [34.73, -29.906, 82.293, -138.378, 59.041, 156.294]
  MoveL 416 to (193.54, -216.3, -12) mm, rotated rx -180 ry 0 rz 179.9 deg; joints [34.721, -29.911, 82.303, -138.39, 59.041, 156.303]
  MoveL 417 to (193.61, -216.02, -12) mm, rotated rx 180 ry 0 rz 179.9 deg; joints [34.712, -29.916, 82.315, -138.402, 59.042, 156.313]
  MoveL 418 to (193.67, -215.71, -12) mm, rotated rx -180 ry 0 rz 179.9 deg; joints [34.702, -29.923, 82.33, -138.416, 59.045, 156.324]
  MoveL 419 to (193.7, -215.4, -12) mm, rotated rx 180 ry 0 rz 179.9 deg; joints [34.693, -29.93, 82.347, -138.429, 59.048, 156.336]
  MoveL 420 to (193.72, -215.09, -12) mm, rotated rx 180 ry 0 rz 179.9 deg; joints [34.684, -29.939, 82.365, -138.443, 59.052, 156.349]
  MoveL 421 to (193.72, -214.79, -12) mm, rotated rx 180 ry 0 rz 179.9 deg; joints [34.676, -29.948, 82.385, -138.456, 59.057, 156.362]
  MoveL 422 to (193.72, 217.86, -12) mm, rotated rx 180 ry 0 rz 179.9 deg; joints [20.946, -39.099, 103.273, -156.79, 65.075, 170.326]
  MoveL 423 to (193.72, 218.16, -12) mm, rotated rx 180 ry 0 rz 179.9 deg; joints [20.935, -39.103, 103.283, -156.803, 65.078, 170.333]
  MoveL 424 to (193.71, 218.32, -12) mm, rotated rx 180 ry 0 rz 179.9 deg; joints [20.93, -39.105, 103.289, -156.81, 65.08, 170.337]
  MoveL 425 to (193.7, 218.47, -12) mm, rotated rx 180 ry 0 rz 179.9 deg; joints [20.925, -39.108, 103.295, -156.816, 65.083, 170.341]
  MoveL 426 to (193.69, 218.62, -12) mm, rotated rx -180 ry 0 rz 179.9 deg; joints [20.919, -39.111, 103.301, -156.823, 65.085, 170.345]
  MoveL 427 to (193.67, 218.78, -12) mm, rotated rx -180 ry 0 rz 179.9 deg; joints [20.914, -39.113, 103.308, -156.829, 65.088, 170.349]
  MoveL 428 to (193.65, 218.93, -12) mm, rotated rx 180 ry 0 rz 179.9 deg; joints [20.909, -39.117, 103.315, -156.836, 65.091, 170.353]
  MoveL 429 to (193.62, 219.08, -12) mm, rotated rx 180 ry 0 rz 179.9 deg; joints [20.904, -39.12, 103.323, -156.842, 65.094, 170.357]
  MoveL 430 to (193.58, 219.24, -12) mm, rotated rx -180 ry 0 rz 179.9 deg; joints [20.899, -39.123, 103.331, -156.848, 65.097, 170.361]
  MoveL 431 to (193.54, 219.39, -12) mm, rotated rx 180 ry 0 rz 179.9 deg; joints [20.894, -39.127, 103.34, -156.854, 65.101, 170.366]
  MoveL 432 to (193.5, 219.54, -12) mm, rotated rx -180 ry 0 rz 179.9 deg; joints [20.889, -39.131, 103.349, -156.861, 65.105, 170.37]
  MoveL 433 to (193.45, 219.7, -12) mm, rotated rx 180 ry 0 rz 179.9 deg; joints [20.884, -39.135, 103.358, -156.867, 65.109, 170.374]
  MoveL 434 to (193.39, 219.85, -12) mm, rotated rx 180 ry 0 rz 179.9 deg; joints [20.879, -39.139, 103.368, -156.873, 65.114, 170.379]
  MoveL 435 to (193.33, 220, -12) mm, rotated rx 180 ry 0 rz 179.9 deg; joints [20.875, -39.143, 103.379, -156.879, 65.118, 170.384]
  MoveL 436 to (193.26, 220.16, -12) mm, rotated rx -180 ry 0 rz 179.9 deg; joints [20.87, -39.148, 103.39, -156.885, 65.123, 170.388]
  MoveL 437 to (193.19, 220.31, -12) mm, rotated rx -180 ry 0 rz 179.9 deg; joints [20.866, -39.153, 103.401, -156.891, 65.129, 170.393]
  MoveL 438 to (193.02, 220.62, -12) mm, rotated rx 180 ry 0 rz 179.9 deg; joints [20.857, -39.164, 103.426, -156.903, 65.14, 170.403]
  MoveL 439 to (192.82, 220.92, -12) mm, rotated rx -180 ry 0 rz 179.9 deg; joints [20.849, -39.175, 103.453, -156.915, 65.153, 170.413]
  MoveL 440 to (192.66, 221.15, -12) mm, rotated rx 180 ry 0 rz 179.9 deg; joints [20.843, -39.185, 103.475, -156.924, 65.164, 170.421]
  MoveL 441 to (192.48, 221.37, -12) mm, rotated rx 180 ry 0 rz 179.9 deg; joints [20.838, -39.195, 103.498, -156.932, 65.175, 170.429]
  MoveL 442 to (192.17, 221.69, -12) mm, rotated rx -180 ry 0 rz 179.9 deg; joints [20.83, -39.211, 103.535, -156.944, 65.193, 170.442]
  MoveL 443 to (191.86, 221.96, -12) mm, rotated rx -180 ry 0 rz 179.9 deg; joints [20.825, -39.226, 103.571, -156.953, 65.211, 170.453]
  MoveL 444 to (191.56, 222.19, -12) mm, rotated rx 180 ry 0 rz 179.9 deg; joints [20.821, -39.241, 103.605, -156.961, 65.228, 170.463]
  MoveL 445 to (191.25, 222.38, -12) mm, rotated rx 180 ry 0 rz 179.9 deg; joints [20.818, -39.255, 103.638, -156.967, 65.245, 170.472]
  MoveL 446 to (190.64, 222.69, -12) mm, rotated rx 180 ry 0 rz 179.9 deg; joints [20.816, -39.282, 103.701, -156.977, 65.278, 170.489]
  MoveL 447 to (190.02, 222.89, -12) mm, rotated rx -180 ry 0 rz 179.9 deg; joints [20.817, -39.308, 103.762, -156.982, 65.309, 170.503]
  MoveL 448 to (189.41, 223.02, -12) mm, rotated rx -180 ry 0 rz 179.9 deg; joints [20.821, -39.333, 103.819, -156.983, 65.34, 170.516]
  MoveL 449 to (188.8, 223.07, -12) mm, rotated rx -180 ry 0 rz 179.9 deg; joints [20.827, -39.357, 103.873, -156.982, 65.369, 170.526]
  MoveL 450 to (187.57, 223.07, -12) mm, rotated rx -180 ry 0 rz 179.9 deg; joints [20.844, -39.403, 103.98, -156.974, 65.428, 170.545]
  MoveL 451 to (-187.57, 223.07, -12) mm, rotated rx 180 ry 0 rz 179.9 deg; joints [27.553, -50.775, 132.624, -152.149, 81.849, 176.414]
  MoveL 452 to (-188.8, 223.05, -12) mm, rotated rx 180 ry 0 rz 179.9 deg; joints [27.582, -50.803, 132.707, -152.123, 81.899, 176.436]
  MoveL 453 to (-189.41, 222.96, -12) mm, rotated rx -180 ry 0 rz 179.9 deg; joints [27.6, -50.816, 132.745, -152.107, 81.923, 176.446]
  MoveL 454 to (-190.02, 222.79, -12) mm, rotated rx -180 ry 0 rz 179.9 deg; joints [27.622, -50.829, 132.781, -152.086, 81.945, 176.454]
  MoveL 455 to (-190.64, 222.53, -12) mm, rotated rx -180 ry 0 rz 179.9 deg; joints [27.648, -50.84, 132.813, -152.062, 81.965, 176.461]
  MoveL 456 to (-191.25, 222.17, -12) mm, rotated rx 180 ry 0 rz 179.9 deg; joints [27.678, -50.85, 132.842, -152.032, 81.983, 176.466]
  MoveL 457 to (-191.56, 221.94, -12) mm, rotated rx 180 ry 0 rz 179.9 deg; joints [27.696, -50.855, 132.854, -152.015, 81.992, 176.468]
  MoveL 458 to (-191.86, 221.66, -12) mm, rotated rx 180 ry 0 rz 179.9 deg; joints [27.715, -50.859, 132.866, -151.996, 81.999, 176.469]
  MoveL 459 to (-192.2, 221.3, -12) mm, rotated rx -180 ry 0 rz 179.9 deg; joints [27.739, -50.862, 132.876, -151.973, 82.006, 176.469]
  MoveL 460 to (-192.48, 220.95, -12) mm, rotated rx 180 ry 0 rz 179.9 deg; joints [27.761, -50.865, 132.882, -151.951, 82.011, 176.468]
  MoveL 461 to (-192.49, 220.92, -12) mm, rotated rx 180 ry 0 rz 179.9 deg; joints [27.762, -50.865, 132.882, -151.949, 82.011, 176.468]
  MoveL 462 to (-192.69, 220.62, -12) mm, rotated rx 180 ry 0 rz 179.9 deg; joints [27.78, -50.866, 132.884, -151.931, 82.013, 176.466]
  MoveL 463 to (-192.86, 220.31, -12) mm, rotated rx -180 ry 0 rz 179.9 deg; joints [27.798, -50.866, 132.885, -151.913, 82.015, 176.464]
  MoveL 464 to (-193, 220, -12) mm, rotated rx -180 ry 0 rz 179.9 deg; joints [27.815, -50.866, 132.883, -151.896, 82.015, 176.461]
  MoveL 465 to (-193.11, 219.7, -12) mm, rotated rx -180 ry 0 rz 179.9 deg; joints [27.831, -50.865, 132.88, -151.88, 82.014, 176.458]
  MoveL 466 to (-193.21, 219.39, -12) mm, rotated rx -180 ry 0 rz 179.9 deg; joints [27.847, -50.864, 132.876, -151.864, 82.012, 176.454]
  MoveL 467 to (-193.28, 219.08, -12) mm, rotated rx -180 ry 0 rz 179.9 deg; joints [27.862, -50.862, 132.87, -151.848, 82.009, 176.451]
  MoveL 468 to (-193.31, 218.93, -12) mm, rotated rx 180 ry 0 rz 179.9 deg; joints [27.87, -50.861, 132.866, -151.84, 82.007, 176.448]
  MoveL 469 to (-193.34, 218.78, -12) mm, rotated rx -180 ry 0 rz 179.9 deg; joints [27.877, -50.86, 132.862, -151.833, 82.006, 176.446]
  MoveL 470 to (-193.36, 218.62, -12) mm, rotated rx -180 ry 0 rz 179.9 deg; joints [27.884, -50.859, 132.858, -151.825, 82.004, 176.444]
  MoveL 471 to (-193.37, 218.47, -12) mm, rotated rx 180 ry 0 rz 179.9 deg; joints [27.892, -50.857, 132.854, -151.818, 82.001, 176.442]
  MoveL 472 to (-193.38, 218.32, -12) mm, rotated rx -180 ry 0 rz 179.9 deg; joints [27.899, -50.856, 132.849, -151.81, 81.999, 176.439]
  MoveL 473 to (-193.39, 218.16, -12) mm, rotated rx -180 ry 0 rz 179.9 deg; joints [27.905, -50.854, 132.844, -151.803, 81.996, 176.437]
  MoveL 474 to (-193.39, 218.01, -12) mm, rotated rx -180 ry 0 rz 179.9 deg; joints [27.912, -50.853, 132.838, -151.796, 81.993, 176.434]
  MoveL 475 to (-193.38, 217.86, -12) mm, rotated rx -180 ry 0 rz 179.9 deg; joints [27.919, -50.851, 132.833, -151.789, 81.99, 176.431]
  MoveL 476 to (-193.37, 217.7, -12) mm, rotated rx -180 ry 0 rz 179.9 deg; joints [27.926, -50.849, 132.826, -151.782, 81.987, 176.429]
  MoveL 477 to (-193.36, 217.55, -12) mm, rotated rx 180 ry 0 rz 179.9 deg; joints [27.932, -50.847, 132.82, -151.775, 81.984, 176.426]
  MoveL 478 to (-193.34, 217.4, -12) mm, rotated rx 180 ry 0 rz 179.9 deg; joints [27.938, -50.845, 132.813, -151.769, 81.98, 176.423]
  MoveL 479 to (-193.32, 217.24, -12) mm, rotated rx 180 ry 0 rz 179.9 deg; joints [27.945, -50.842, 132.806, -151.762, 81.976, 176.42]
  MoveL 480 to (-192.47, 211.92, -12) mm, rotated rx -180 ry 0 rz 179.9 deg; joints [28.159, -50.761, 132.557, -151.534, 81.842, 176.312]
  MoveL 481 to (-126.12, -206.86, -12) mm, rotated rx 180 ry 0 rz 179.9 deg; joints [41.666, -41.498, 108.14, -135.624, 71.876, 164.113]
  MoveL 482 to (-126.05, -207.32, -12) mm, rotated rx -180 ry 0 rz 179.9 deg; joints [41.678, -41.484, 108.108, -135.608, 71.866, 164.095]
  MoveC 483 to (-126.68, -208.41, -12) mm, rotated rx 180 ry 0 rz 179.9 deg; joints [41.727, -41.475, 108.085, -135.556, 71.869, 164.071] to (-127.87, -208.02, -12) mm, rotated rx 180 ry 0 rz 179.9 deg; joints [41.747, -41.519, 108.188, -135.549, 71.917, 164.108]
  MoveL 484 to (-128.72, -206.73, -12) mm, rotated rx -180 ry 0 rz 179.9 deg; joints [41.731, -41.576, 108.321, -135.583, 71.968, 164.17]
  Set speed (5.6 mm/s)
  MoveL 485 to (-128.72, -206.73, -17) mm, rotated rx -180 ry 0 rz 179.9 deg; joints [41.734, -41.292, 108.271, -135.633, 72.134, 164.34]
  MoveC 486 to (-128.43, -206.68, -17.71) mm, rotated rx -180 ry 0 rz 179.9 deg; joints [41.725, -41.245, 108.247, -135.646, 72.149, 164.359] to (-127.73, -206.57, -18) mm, rotated rx -180 ry 0 rz 179.9 deg; joints [41.704, -41.211, 108.204, -135.666, 72.136, 164.359]
  Set speed (16.7 mm/s)
  MoveC 487 to (-126.98, -206.75, -18) mm, rotated rx -180 ry 0 rz 179.9 deg; joints [41.689, -41.186, 108.143, -135.673, 72.107, 164.338] to (-126.58, -207.4, -18) mm, rotated rx 180 ry 0 rz 179.9 deg; joints [41.698, -41.158, 108.078, -135.656, 72.083, 164.307]
  MoveL 488 to (-124.73, -219.08, -18) mm, rotated rx 180 ry 0 rz 179.9 deg; joints [41.993, -40.816, 107.253, -135.248, 71.821, 163.864]
  MoveL 489 to (-124.68, -219.39, -18) mm, rotated rx 180 ry 0 rz 179.9 deg; joints [42, -40.806, 107.231, -135.237, 71.814, 163.852]
  MoveL 490 to (-124.61, -219.7, -18) mm, rotated rx -180 ry 0 rz 179.9 deg; joints [42.007, -40.797, 107.208, -135.227, 71.806, 163.84]
  MoveL 491 to (-124.52, -220, -18) mm, rotated rx 180 ry 0 rz 179.9 deg; joints [42.014, -40.786, 107.183, -135.217, 71.798, 163.828]
  MoveL 492 to (-124.41, -220.31, -18) mm, rotated rx -180 ry 0 rz 179.9 deg; joints [42.02, -40.776, 107.157, -135.207, 71.789, 163.815]
  MoveL 493 to (-124.28, -220.62, -18) mm, rotated rx 180 ry 0 rz 179.9 deg; joints [42.025, -40.764, 107.13, -135.198, 71.779, 163.801]
  MoveL 494 to (-124.12, -220.92, -18) mm, rotated rx -180 ry 0 rz 179.9 deg; joints [42.03, -40.752, 107.1, -135.189, 71.769, 163.787]
  MoveL 495 to (-123.98, -221.16, -18) mm, rotated rx -180 ry 0 rz 179.9 deg; joints [42.033, -40.742, 107.077, -135.183, 71.76, 163.776]
  MoveL 496 to (-123.82, -221.39, -18) mm, rotated rx -180 ry 0 rz 179.9 deg; joints [42.036, -40.732, 107.053, -135.177, 71.751, 163.765]
  MoveL 497 to (-123.69, -221.56, -18) mm, rotated rx -180 ry 0 rz 179.9 deg; joints [42.037, -40.723, 107.033, -135.173, 71.743, 163.756]
  MoveL 498 to (-123.54, -221.74, -18) mm, rotated rx 180 ry 0 rz 179.9 deg; joints [42.039, -40.715, 107.013, -135.169, 71.735, 163.747]
  MoveL 499 to (-123.38, -221.91, -18) mm, rotated rx 180 ry 0 rz 179.9 deg; joints [42.04, -40.706, 106.992, -135.165, 71.727, 163.738]
  MoveL 500 to (-123.21, -222.09, -18) mm, rotated rx -180 ry 0 rz 179.9 deg; joints [42.04, -40.696, 106.969, -135.162, 71.718, 163.728]
  MoveL 501 to (-122.9, -222.35, -18) mm, rotated rx -180 ry 0 rz 179.9 deg; joints [42.04, -40.681, 106.933, -135.157, 71.703, 163.712]
  MoveL 502 to (-122.6, -222.58, -18) mm, rotated rx 180 ry 0 rz 179.9 deg; joints [42.038, -40.666, 106.898, -135.154, 71.688, 163.698]
  MoveL 503 to (-122.29, -222.77, -18) mm, rotated rx -180 ry 0 rz 179.9 deg; joints [42.036, -40.652, 106.866, -135.152, 71.674, 163.685]
  MoveL 504 to (-121.98, -222.94, -18) mm, rotated rx -180 ry 0 rz 179.9 deg; joints [42.033, -40.639, 106.835, -135.151, 71.661, 163.673]
  MoveL 505 to (-121.68, -223.08, -18) mm, rotated rx -180 ry 0 rz 179.9 deg; joints [42.029, -40.627, 106.806, -135.151, 71.648, 163.662]
  MoveL 506 to (-121.37, -223.19, -18) mm, rotated rx -180 ry 0 rz 179.9 deg; joints [42.024, -40.615, 106.779, -135.152, 71.635, 163.651]
  MoveL 507 to (-121, -223.3, -18) mm, rotated rx 180 ry 0 rz 179.9 deg; joints [42.017, -40.602, 106.747, -135.155, 71.621, 163.64]
  MoveL 508 to (-120.63, -223.38, -18) mm, rotated rx 180 ry 0 rz 179.9 deg; joints [42.01, -40.589, 106.718, -135.158, 71.607, 163.63]
  MoveL 509 to (-120.2, -223.44, -18) mm, rotated rx -180 ry 0 rz 179.9 deg; joints [42, -40.575, 106.686, -135.164, 71.591, 163.619]
  MoveL 510 to (-119.78, -223.45, -18) mm, rotated rx -180 ry 0 rz 179.9 deg; joints [41.989, -40.562, 106.656, -135.171, 71.576, 163.609]
  MoveL 511 to (188.58, -223.45, -18) mm, rotated rx -180 ry 0 rz 179.9 deg; joints [35.016, -29.631, 82.237, -138.16, 59.32, 156.312]
  MoveL 512 to (189.08, -223.44, -18) mm, rotated rx 180 ry 0 rz 179.9 deg; joints [35.006, -29.609, 82.19, -138.161, 59.298, 156.298]
  MoveL 513 to (189.33, -223.42, -18) mm, rotated rx 180 ry 0 rz 179.9 deg; joints [35.001, -29.599, 82.168, -138.162, 59.286, 156.292]
  MoveL 514 to (189.58, -223.38, -18) mm, rotated rx -180 ry 0 rz 179.9 deg; joints [34.995, -29.589, 82.147, -138.164, 59.276, 156.286]
  MoveL 515 to (190.02, -223.28, -18) mm, rotated rx 180 ry 0 rz 179.9 deg; joints [34.984, -29.573, 82.112, -138.168, 59.257, 156.277]
  MoveL 516 to (190.33, -223.19, -18) mm, rotated rx -180 ry 0 rz 179.9 deg; joints [34.975, -29.563, 82.089, -138.172, 59.244, 156.272]
  MoveL 517 to (190.64, -223.07, -18) mm, rotated rx -180 ry 0 rz 179.9 deg; joints [34.966, -29.553, 82.068, -138.178, 59.232, 156.268]
  MoveL 518 to (190.94, -222.93, -18) mm, rotated rx 180 ry 0 rz 179.9 deg; joints [34.956, -29.544, 82.048, -138.184, 59.22, 156.265]
  MoveL 519 to (191.25, -222.77, -18) mm, rotated rx -180 ry 0 rz 179.9 deg; joints [34.946, -29.535, 82.03, -138.191, 59.209, 156.263]
  MoveL 520 to (191.56, -222.57, -18) mm, rotated rx 180 ry 0 rz 179.9 deg; joints [34.935, -29.528, 82.014, -138.2, 59.198, 156.263]
  MoveL 521 to (191.86, -222.34, -18) mm, rotated rx 180 ry 0 rz 179.9 deg; joints [34.922, -29.521, 82, -138.21, 59.188, 156.263]
  MoveL 522 to (192.17, -222.08, -18) mm, rotated rx -180 ry 0 rz 179.9 deg; joints [34.909, -29.516, 81.989, -138.222, 59.178, 156.266]
  MoveL 523 to (192.33, -221.92, -18) mm, rotated rx -180 ry 0 rz 179.9 deg; joints [34.902, -29.513, 81.984, -138.229, 59.173, 156.268]
  MoveL 524 to (192.48, -221.76, -18) mm, rotated rx 180 ry 0 rz 179.9 deg; joints [34.894, -29.512, 81.981, -138.236, 59.169, 156.27]
  MoveL 525 to (192.65, -221.55, -18) mm, rotated rx 180 ry 0 rz 179.9 deg; joints [34.885, -29.51, 81.978, -138.245, 59.164, 156.274]
  MoveL 526 to (192.8, -221.34, -18) mm, rotated rx -180 ry 0 rz 179.9 deg; joints [34.877, -29.51, 81.977, -138.254, 59.16, 156.278]
  MoveL 527 to (192.94, -221.13, -18) mm, rotated rx -180 ry 0 rz 179.9 deg; joints [34.868, -29.51, 81.978, -138.263, 59.157, 156.283]
  MoveL 528 to (193.07, -220.92, -18) mm, rotated rx 180 ry 0 rz 179.9 deg; joints [34.86, -29.511, 81.98, -138.272, 59.155, 156.288]
  MoveL 529 to (193.23, -220.62, -18) mm, rotated rx -180 ry 0 rz 179.9 deg; joints [34.849, -29.513, 81.985, -138.286, 59.152, 156.297]
  MoveL 530 to (193.36, -220.31, -18) mm, rotated rx 180 ry 0 rz 179.9 deg; joints [34.837, -29.516, 81.992, -138.299, 59.151, 156.306]
  MoveL 531 to (193.47, -220, -18) mm, rotated rx -180 ry 0 rz 179.9 deg; joints [34.827, -29.52, 82.002, -138.312, 59.151, 156.316]
  MoveL 532 to (193.56, -219.7, -18) mm, rotated rx -180 ry 0 rz 179.9 deg; joints [34.817, -29.526, 82.014, -138.326, 59.152, 156.326]
  MoveL 533 to (193.63, -219.39, -18) mm, rotated rx 180 ry 0 rz 179.9 deg; joints [34.807, -29.532, 82.028, -138.339, 59.153, 156.337]
  MoveL 534 to (193.68, -219.08, -18) mm, rotated rx 180 ry 0 rz 179.9 deg; joints [34.798, -29.539, 82.043, -138.353, 59.156, 156.349]
  MoveL 535 to (193.71, -218.78, -18) mm, rotated rx -180 ry 0 rz 179.9 deg; joints [34.789, -29.547, 82.061, -138.366, 59.159, 156.361]
  MoveL 536 to (193.72, -218.47, -18) mm, rotated rx 180 ry 0 rz 179.9 deg; joints [34.78, -29.555, 82.08, -138.38, 59.164, 156.374]
  MoveL 537 to (193.72, 219.7, -18) mm, rotated rx -180 ry 0 rz 179.9 deg; joints [20.883, -38.799, 103.273, -156.914, 65.34, 170.484]
  MoveL 538 to (193.71, 220, -18) mm, rotated rx -180 ry 0 rz 179.9 deg; joints [20.872, -38.803, 103.284, -156.927, 65.344, 170.491]
  MoveL 539 to (193.68, 220.31, -18) mm, rotated rx 180 ry 0 rz 179.9 deg; joints [20.861, -38.809, 103.297, -156.94, 65.349, 170.499]
  MoveL 540 to (193.62, 220.62, -18) mm, rotated rx 180 ry 0 rz 179.9 deg; joints [20.851, -38.815, 103.312, -156.952, 65.355, 170.507]
  MoveL 541 to (193.55, 220.92, -18) mm, rotated rx 180 ry 0 rz 179.9 deg; joints [20.841, -38.822, 103.328, -156.965, 65.362, 170.516]
  MoveL 542 to (193.48, 221.18, -18) mm, rotated rx 180 ry 0 rz 179.9 deg; joints [20.833, -38.828, 103.343, -156.975, 65.369, 170.523]
  MoveL 543 to (193.39, 221.43, -18) mm, rotated rx -180 ry 0 rz 179.9 deg; joints [20.825, -38.835, 103.359, -156.985, 65.376, 170.53]
  MoveL 544 to (193.29, 221.68, -18) mm, rotated rx 180 ry 0 rz 179.9 deg; joints [20.818, -38.842, 103.377, -156.995, 65.384, 170.538]
  MoveL 545 to (193.16, 221.93, -18) mm, rotated rx 180 ry 0 rz 179.9 deg; joints [20.81, -38.85, 103.396, -157.005, 65.393, 170.546]
  MoveL 546 to (193.02, 222.19, -18) mm, rotated rx -180 ry 0 rz 179.9 deg; joints [20.803, -38.859, 103.416, -157.015, 65.402, 170.554]
  MoveL 547 to (192.87, 222.44, -18) mm, rotated rx 180 ry 0 rz 179.9 deg; joints [20.796, -38.869, 103.438, -157.025, 65.413, 170.562]
  MoveL 548 to (192.68, 222.69, -18) mm, rotated rx 180 ry 0 rz 179.9 deg; joints [20.79, -38.879, 103.463, -157.034, 65.425, 170.571]
  MoveL 549 to (192.48, 222.94, -18) mm, rotated rx 180 ry 0 rz 179.9 deg; joints [20.783, -38.89, 103.489, -157.044, 65.438, 170.58]
  MoveL 550 to (192.27, 223.16, -18) mm, rotated rx 180 ry 0 rz 179.9 deg; joints [20.778, -38.901, 103.514, -157.052, 65.45, 170.589]
  MoveL 551 to (192.04, 223.38, -18) mm, rotated rx -180 ry 0 rz 179.9 deg; joints [20.774, -38.912, 103.541, -157.06, 65.463, 170.597]
  MoveL 552 to (191.79, 223.59, -18) mm, rotated rx -180 ry 0 rz 179.9 deg; joints [20.77, -38.925, 103.57, -157.067, 65.478, 170.606]
  MoveL 553 to (191.54, 223.77, -18) mm, rotated rx -180 ry 0 rz 179.9 deg; joints [20.767, -38.937, 103.598, -157.073, 65.492, 170.614]
  MoveL 554 to (191.28, 223.93, -18) mm, rotated rx -180 ry 0 rz 179.9 deg; joints [20.764, -38.948, 103.625, -157.078, 65.506, 170.622]
  MoveL 555 to (191.03, 224.08, -18) mm, rotated rx 180 ry 0 rz 179.9 deg; joints [20.763, -38.96, 103.652, -157.083, 65.52, 170.629]
  MoveL 556 to (190.78, 224.2, -18) mm, rotated rx -180 ry 0 rz 179.9 deg; joints [20.762, -38.971, 103.678, -157.087, 65.533, 170.636]
  MoveL 557 to (190.53, 224.3, -18) mm, rotated rx 180 ry 0 rz 179.9 deg; joints [20.761, -38.982, 103.703, -157.09, 65.547, 170.642]
  MoveL 558 to (190.28, 224.39, -18) mm, rotated rx -180 ry 0 rz 179.9 deg; joints [20.761, -38.992, 103.728, -157.092, 65.56, 170.648]
  MoveL 559 to (190.02, 224.47, -18) mm, rotated rx -180 ry 0 rz 179.9 deg; joints [20.762, -39.003, 103.752, -157.093, 65.573, 170.654]
  MoveL 560 to (189.72, 224.54, -18) mm, rotated rx 180 ry 0 rz 179.9 deg; joints [20.764, -39.015, 103.781, -157.095, 65.588, 170.66]
  MoveL 561 to (189.41, 224.59, -18) mm, rotated rx 180 ry 0 rz 179.9 deg; joints [20.766, -39.027, 103.809, -157.095, 65.603, 170.666]
  MoveL 562 to (189.1, 224.63, -18) mm, rotated rx -180 ry 0 rz 179.9 deg; joints [20.769, -39.039, 103.837, -157.095, 65.618, 170.672]
  MoveL 563 to (188.8, 224.64, -18) mm, rotated rx 180 ry 0 rz 179.9 deg; joints [20.773, -39.051, 103.864, -157.093, 65.633, 170.677]
  MoveL 564 to (187.57, 224.64, -18) mm, rotated rx -180 ry 0 rz 179.9 deg; joints [20.79, -39.097, 103.97, -157.086, 65.692, 170.695]
  MoveL 565 to (-182.67, 224.64, -18) mm, rotated rx -180 ry 0 rz 179.9 deg; joints [27.373, -50.225, 132.273, -152.343, 82.014, 176.53]
  MoveL 566 to (-188.8, 224.64, -18) mm, rotated rx -180 ry 0 rz 179.9 deg; joints [27.515, -50.366, 132.691, -152.218, 82.268, 176.643]
  MoveL 567 to (-189.1, 224.63, -18) mm, rotated rx -180 ry 0 rz 179.9 deg; joints [27.523, -50.372, 132.711, -152.211, 82.28, 176.649]
  MoveL 568 to (-189.41, 224.59, -18) mm, rotated rx 180 ry 0 rz 179.9 deg; joints [27.531, -50.379, 132.731, -152.204, 82.292, 176.654]
  MoveL 569 to (-189.72, 224.54, -18) mm, rotated rx 180 ry 0 rz 179.9 deg; joints [27.541, -50.385, 132.75, -152.195, 82.304, 176.659]
  MoveL 570 to (-190.02, 224.47, -18) mm, rotated rx -180 ry 0 rz 179.9 deg; joints [27.551, -50.392, 132.768, -152.185, 82.315, 176.663]
  MoveL 571 to (-190.28, 224.39, -18) mm, rotated rx 180 ry 0 rz 179.9 deg; joints [27.56, -50.397, 132.782, -152.177, 82.324, 176.666]
  MoveL 572 to (-190.53, 224.3, -18) mm, rotated rx 180 ry 0 rz 179.9 deg; joints [27.57, -50.401, 132.796, -152.167, 82.333, 176.67]
  MoveL 573 to (-190.78, 224.2, -18) mm, rotated rx -180 ry 0 rz 179.9 deg; joints [27.581, -50.406, 132.81, -152.157, 82.341, 176.672]
  MoveL 574 to (-191.03, 224.08, -18) mm, rotated rx 180 ry 0 rz 179.9 deg; joints [27.592, -50.41, 132.823, -152.146, 82.349, 176.675]
  MoveL 575 to (-191.28, 223.93, -18) mm, rotated rx 180 ry 0 rz 179.9 deg; joints [27.604, -50.414, 132.835, -152.135, 82.357, 176.677]
  MoveL 576 to (-191.54, 223.77, -18) mm, rotated rx -180 ry 0 rz 179.9 deg; joints [27.617, -50.418, 132.846, -152.122, 82.364, 176.679]
  MoveL 577 to (-191.79, 223.59, -18) mm, rotated rx -180 ry 0 rz 179.9 deg; joints [27.631, -50.422, 132.857, -152.108, 82.371, 176.681]
  MoveL 578 to (-192.04, 223.38, -18) mm, rotated rx -180 ry 0 rz 179.9 deg; joints [27.646, -50.426, 132.866, -152.093, 82.378, 176.682]
  MoveL 579 to (-192.27, 223.16, -18) mm, rotated rx -180 ry 0 rz 179.9 deg; joints [27.661, -50.428, 132.874, -152.079, 82.383, 176.683]
  MoveL 580 to (-192.47, 222.94, -18) mm, rotated rx 180 ry 0 rz 179.9 deg; joints [27.676, -50.431, 132.88, -152.064, 82.388, 176.683]
  MoveL 581 to (-192.68, 222.69, -18) mm, rotated rx -180 ry 0 rz 179.9 deg; joints [27.692, -50.433, 132.885, -152.048, 82.391, 176.683]
  MoveL 582 to (-192.86, 222.44, -18) mm, rotated rx 180 ry 0 rz 179.9 deg; joints [27.707, -50.434, 132.889, -152.033, 82.394, 176.682]
  MoveL 583 to (-193.02, 222.19, -18) mm, rotated rx 180 ry 0 rz 179.9 deg; joints [27.722, -50.435, 132.891, -152.018, 82.396, 176.68]
  MoveL 584 to (-193.16, 221.93, -18) mm, rotated rx -180 ry 0 rz 179.9 deg; joints [27.737, -50.435, 132.891, -152.003, 82.397, 176.679]
  MoveL 585 to (-193.29, 221.68, -18) mm, rotated rx 180 ry 0 rz 179.9 deg; joints [27.751, -50.435, 132.89, -151.989, 82.397, 176.677]
  MoveL 586 to (-193.39, 221.43, -18) mm, rotated rx 180 ry 0 rz 179.9 deg; joints [27.764, -50.435, 132.888, -151.975, 82.397, 176.674]
  MoveL 587 to (-193.48, 221.18, -18) mm, rotated rx 180 ry 0 rz 179.9 deg; joints [27.778, -50.434, 132.885, -151.962, 82.395, 176.672]
  MoveL 588 to (-193.55, 220.92, -18) mm, rotated rx -180 ry 0 rz 179.9 deg; joints [27.79, -50.433, 132.881, -151.949, 82.394, 176.669]
  MoveL 589 to (-193.62, 220.62, -18) mm, rotated rx 180 ry 0 rz 179.9 deg; joints [27.806, -50.431, 132.875, -151.933, 82.391, 176.665]
  MoveL 590 to (-193.68, 220.31, -18) mm, rotated rx -180 ry 0 rz 179.9 deg; joints [27.821, -50.429, 132.868, -151.918, 82.387, 176.661]
  MoveL 591 to (-193.71, 220, -18) mm, rotated rx -180 ry 0 rz 179.9 deg; joints [27.835, -50.426, 132.859, -151.903, 82.383, 176.656]
  MoveL 592 to (-193.72, 219.7, -18) mm, rotated rx -180 ry 0 rz 179.9 deg; joints [27.849, -50.423, 132.849, -151.889, 82.377, 176.651]
  MoveL 593 to (-193.72, 216.63, -18) mm, rotated rx -180 ry 0 rz 179.9 deg; joints [27.984, -50.389, 132.739, -151.747, 82.319, 176.599]
  MoveL 594 to (-193.71, 216.32, -18) mm, rotated rx 180 ry 0 rz 179.9 deg; joints [27.998, -50.385, 132.727, -151.733, 82.313, 176.594]
  MoveL 595 to (-193.67, 216.02, -18) mm, rotated rx -180 ry 0 rz 179.9 deg; joints [28.01, -50.381, 132.714, -151.72, 82.305, 176.588]
  MoveL 596 to (-193.29, 213.56, -18) mm, rotated rx 180 ry 0 rz 179.9 deg; joints [28.109, -50.345, 132.599, -151.615, 82.243, 176.539]
  MoveL 597 to (-192.47, 208.44, -18) mm, rotated rx 180 ry 0 rz 179.9 deg; joints [28.315, -50.268, 132.358, -151.397, 82.112, 176.435]
  MoveL 598 to (-126.66, -206.94, -18) mm, rotated rx -180 ry 0 rz 179.9 deg; joints [41.686, -41.171, 108.11, -135.671, 72.093, 164.324]
  MoveL 599 to (-126.58, -207.4, -18) mm, rotated rx 180 ry 0 rz 179.9 deg; joints [41.698, -41.158, 108.078, -135.656, 72.083, 164.307]
  MoveC 600 to (-127.33, -208.53, -18) mm, rotated rx -180 ry 0 rz 179.9 deg; joints [41.751, -41.152, 108.06, -135.599, 72.089, 164.283] to (-128.52, -207.88, -18) mm, rotated rx -180 ry 0 rz 179.9 deg; joints [41.763, -41.202, 108.178, -135.602, 72.141, 164.33]
  MoveL 601 to (-128.9, -206.76, -18) mm, rotated rx 180 ry 0 rz 179.9 deg; joints [41.74, -41.24, 108.271, -135.638, 72.174, 164.376]
  Set speed (5.6 mm/s)
  MoveL 602 to (-128.9, -206.76, -19.05) mm, rotated rx 180 ry 0 rz 179.9 deg; joints [41.741, -41.181, 108.26, -135.648, 72.208, 164.412]
  MoveC 603 to (-128.61, -206.71, -19.76) mm, rotated rx 180 ry 0 rz 179.9 deg; joints [41.732, -41.133, 108.236, -135.662, 72.223, 164.431] to (-127.91, -206.6, -20.05) mm, rotated rx -180 ry 0 rz 179.9 deg; joints [41.71, -41.099, 108.193, -135.682, 72.21, 164.431]
  Set speed (16.7 mm/s)
  MoveL 604 to (-126.77, -207.43, -20.05) mm, rotated rx 180 ry 0 rz 179.9 deg; joints [41.705, -41.046, 108.066, -135.671, 72.156, 164.379]
  MoveL 605 to (-124.73, -220.31, -20.05) mm, rotated rx 180 ry 0 rz 179.9 deg; joints [42.029, -40.669, 107.157, -135.222, 71.867, 163.89]
  MoveL 606 to (-124.67, -220.62, -20.05) mm, rotated rx 180 ry 0 rz 179.9 deg; joints [42.037, -40.66, 107.135, -135.212, 71.86, 163.878]
  MoveL 607 to (-124.6, -220.92, -20.05) mm, rotated rx 180 ry 0 rz 179.9 deg; joints [42.044, -40.65, 107.111, -135.201, 71.852, 163.866]
  MoveL 608 to (-124.54, -221.13, -20.05) mm, rotated rx 180 ry 0 rz 179.9 deg; joints [42.048, -40.644, 107.095, -135.195, 71.847, 163.858]
  MoveL 609 to (-124.47, -221.34, -20.05) mm, rotated rx -180 ry 0 rz 179.9 deg; joints [42.053, -40.636, 107.078, -135.188, 71.841, 163.849]
  MoveL 610 to (-124.39, -221.54, -20.05) mm, rotated rx 180 ry 0 rz 179.9 deg; joints [42.057, -40.629, 107.06, -135.182, 71.835, 163.84]
  MoveL 611 to (-124.3, -221.75, -20.05) mm, rotated rx -180 ry 0 rz 179.9 deg; joints [42.06, -40.621, 107.042, -135.176, 71.828, 163.831]
  MoveL 612 to (-124.2, -221.95, -20.05) mm, rotated rx -180 ry 0 rz 179.9 deg; joints [42.063, -40.613, 107.023, -135.17, 71.821, 163.822]
  MoveL 613 to (-124.09, -222.16, -20.05) mm, rotated rx -180 ry 0 rz 179.9 deg; joints [42.066, -40.605, 107.003, -135.164, 71.814, 163.813]
  MoveL 614 to (-123.96, -222.36, -20.05) mm, rotated rx 180 ry 0 rz 179.9 deg; joints [42.069, -40.596, 106.982, -135.159, 71.806, 163.803]
  MoveL 615 to (-123.82, -222.57, -20.05) mm, rotated rx -180 ry 0 rz 179.9 deg; joints [42.071, -40.587, 106.96, -135.153, 71.797, 163.793]
  MoveL 616 to (-123.67, -222.77, -20.05) mm, rotated rx -180 ry 0 rz 179.9 deg; joints [42.073, -40.577, 106.937, -135.148, 71.789, 163.782]
  MoveL 617 to (-123.49, -222.97, -20.05) mm, rotated rx 180 ry 0 rz 179.9 deg; joints [42.075, -40.567, 106.913, -135.144, 71.779, 163.772]
  MoveL 618 to (-123.29, -223.19, -20.05) mm, rotated rx 180 ry 0 rz 179.9 deg; joints [42.075, -40.556, 106.886, -135.139, 71.768, 163.76]
  MoveL 619 to (-123.09, -223.38, -20.05) mm, rotated rx -180 ry 0 rz 179.9 deg; joints [42.076, -40.545, 106.861, -135.136, 71.758, 163.749]
  MoveL 620 to (-122.87, -223.56, -20.05) mm, rotated rx 180 ry 0 rz 179.9 deg; joints [42.075, -40.535, 106.836, -135.133, 71.748, 163.738]
  MoveL 621 to (-122.66, -223.72, -20.05) mm, rotated rx -180 ry 0 rz 179.9 deg; joints [42.074, -40.524, 106.812, -135.131, 71.738, 163.728]
  MoveL 622 to (-122.44, -223.86, -20.05) mm, rotated rx 180 ry 0 rz 179.9 deg; joints [42.073, -40.515, 106.789, -135.129, 71.728, 163.719]
  MoveL 623 to (-122.23, -223.99, -20.05) mm, rotated rx -180 ry 0 rz 179.9 deg; joints [42.071, -40.505, 106.766, -135.128, 71.718, 163.71]
  MoveL 624 to (-122.01, -224.11, -20.05) mm, rotated rx -180 ry 0 rz 179.9 deg; joints [42.068, -40.496, 106.745, -135.127, 71.709, 163.702]
  MoveL 625 to (-121.8, -224.21, -20.05) mm, rotated rx 180 ry 0 rz 179.9 deg; joints [42.066, -40.487, 106.725, -135.127, 71.7, 163.694]
  MoveL 626 to (-121.37, -224.37, -20.05) mm, rotated rx -180 ry 0 rz 179.9 deg; joints [42.059, -40.471, 106.686, -135.129, 71.682, 163.679]
  MoveL 627 to (-121.06, -224.47, -20.05) mm, rotated rx 180 ry 0 rz 179.9 deg; joints [42.054, -40.46, 106.659, -135.131, 71.67, 163.669]
  MoveL 628 to (-120.76, -224.54, -20.05) mm, rotated rx 180 ry 0 rz 179.9 deg; joints [42.048, -40.449, 106.634, -135.133, 71.658, 163.661]
  MoveL 629 to (-120.45, -224.59, -20.05) mm, rotated rx 180 ry 0 rz 179.9 deg; joints [42.041, -40.439, 106.611, -135.137, 71.646, 163.652]
  MoveL 630 to (-120.14, -224.62, -20.05) mm, rotated rx 180 ry 0 rz 179.9 deg; joints [42.034, -40.429, 106.588, -135.141, 71.635, 163.645]
  MoveL 631 to (-118.92, -224.64, -20.05) mm, rotated rx 180 ry 0 rz 179.9 deg; joints [42.002, -40.393, 106.505, -135.162, 71.592, 163.619]
  MoveL 632 to (182.67, -224.64, -20.05) mm, rotated rx -180 ry 0 rz 179.9 deg; joints [35.165, -29.754, 82.691, -138.133, 59.627, 156.491]
  MoveL 633 to (188.8, -224.64, -20.05) mm, rotated rx 180 ry 0 rz 179.9 deg; joints [35.046, -29.489, 82.116, -138.137, 59.347, 156.313]
  MoveL 634 to (189.1, -224.62, -20.05) mm, rotated rx 180 ry 0 rz 179.9 deg; joints [35.039, -29.476, 82.088, -138.138, 59.334, 156.304]
  MoveL 635 to (189.41, -224.59, -20.05) mm, rotated rx 180 ry 0 rz 179.9 deg; joints [35.032, -29.464, 82.061, -138.14, 59.32, 156.297]
  MoveL 636 to (189.72, -224.54, -20.05) mm, rotated rx 180 ry 0 rz 179.9 deg; joints [35.025, -29.452, 82.035, -138.142, 59.307, 156.29]
  MoveL 637 to (190.02, -224.46, -20.05) mm, rotated rx 180 ry 0 rz 179.9 deg; joints [35.017, -29.441, 82.011, -138.145, 59.294, 156.284]
  MoveL 638 to (190.27, -224.39, -20.05) mm, rotated rx -180 ry 0 rz 179.9 deg; joints [35.01, -29.432, 81.992, -138.149, 59.284, 156.28]
  MoveL 639 to (190.53, -224.3, -20.05) mm, rotated rx -180 ry 0 rz 179.9 deg; joints [35.003, -29.424, 81.975, -138.153, 59.274, 156.276]
  MoveL 640 to (190.78, -224.19, -20.05) mm, rotated rx 180 ry 0 rz 179.9 deg; joints [34.995, -29.416, 81.958, -138.157, 59.264, 156.273]
  MoveL 641 to (191.03, -224.07, -20.05) mm, rotated rx 180 ry 0 rz 179.9 deg; joints [34.987, -29.409, 81.942, -138.163, 59.254, 156.271]
  MoveL 642 to (191.28, -223.93, -20.05) mm, rotated rx 180 ry 0 rz 179.9 deg; joints [34.978, -29.402, 81.928, -138.169, 59.245, 156.27]
  MoveL 643 to (191.53, -223.77, -20.05) mm, rotated rx -180 ry 0 rz 179.9 deg; joints [34.969, -29.396, 81.914, -138.176, 59.236, 156.269]
  MoveL 644 to (191.78, -223.59, -20.05) mm, rotated rx -180 ry 0 rz 179.9 deg; joints [34.959, -29.39, 81.903, -138.184, 59.227, 156.27]
  MoveL 645 to (192.04, -223.38, -20.05) mm, rotated rx -180 ry 0 rz 179.9 deg; joints [34.948, -29.386, 81.893, -138.193, 59.219, 156.271]
  MoveL 646 to (192.27, -223.16, -20.05) mm, rotated rx 180 ry 0 rz 179.9 deg; joints [34.938, -29.382, 81.885, -138.203, 59.212, 156.274]
  MoveL 647 to (192.48, -222.94, -20.05) mm, rotated rx 180 ry 0 rz 179.9 deg; joints [34.928, -29.38, 81.88, -138.213, 59.206, 156.277]
  MoveL 648 to (192.68, -222.69, -20.05) mm, rotated rx 180 ry 0 rz 179.9 deg; joints [34.917, -29.378, 81.877, -138.224, 59.2, 156.282]
  MoveL 649 to (192.86, -222.44, -20.05) mm, rotated rx -180 ry 0 rz 179.9 deg; joints [34.906, -29.378, 81.877, -138.235, 59.196, 156.287]
  MoveL 650 to (193.02, -222.18, -20.05) mm, rotated rx -180 ry 0 rz 179.9 deg; joints [34.896, -29.378, 81.878, -138.246, 59.193, 156.293]
  MoveL 651 to (193.16, -221.93, -20.05) mm, rotated rx 180 ry 0 rz 179.9 deg; joints [34.887, -29.38, 81.882, -138.257, 59.19, 156.3]
  MoveL 652 to (193.28, -221.68, -20.05) mm, rotated rx 180 ry 0 rz 179.9 deg; joints [34.878, -29.382, 81.887, -138.268, 59.189, 156.307]
  MoveL 653 to (193.39, -221.43, -20.05) mm, rotated rx 180 ry 0 rz 179.9 deg; joints [34.869, -29.385, 81.894, -138.279, 59.188, 156.315]
  MoveL 654 to (193.48, -221.18, -20.05) mm, rotated rx 180 ry 0 rz 179.9 deg; joints [34.86, -29.388, 81.902, -138.29, 59.188, 156.323]
  MoveL 655 to (193.55, -220.92, -20.05) mm, rotated rx -180 ry 0 rz 179.9 deg; joints [34.852, -29.393, 81.911, -138.301, 59.189, 156.331]
  MoveL 656 to (193.62, -220.62, -20.05) mm, rotated rx -180 ry 0 rz 179.9 deg; joints [34.842, -29.399, 81.925, -138.314, 59.19, 156.342]
  MoveL 657 to (193.67, -220.31, -20.05) mm, rotated rx -180 ry 0 rz 179.9 deg; joints [34.832, -29.406, 81.94, -138.328, 59.193, 156.354]
  MoveL 658 to (193.71, -220, -20.05) mm, rotated rx 180 ry 0 rz 179.9 deg; joints [34.823, -29.413, 81.957, -138.341, 59.196, 156.366]
  MoveL 659 to (193.72, -219.7, -20.05) mm, rotated rx 180 ry 0 rz 179.9 deg; joints [34.815, -29.422, 81.976, -138.355, 59.2, 156.379]
  MoveL 660 to (193.72, 219.7, -20.05) mm, rotated rx 180 ry 0 rz 179.9 deg; joints [20.883, -38.687, 103.252, -156.929, 65.423, 170.522]
  MoveL 661 to (193.71, 220, -20.05) mm, rotated rx 180 ry 0 rz 179.9 deg; joints [20.873, -38.692, 103.263, -156.942, 65.427, 170.53]
  MoveL 662 to (193.68, 220.31, -20.05) mm, rotated rx -180 ry 0 rz 179.9 deg; joints [20.862, -38.697, 103.276, -156.955, 65.432, 170.537]
  MoveL 663 to (193.62, 220.62, -20.05) mm, rotated rx -180 ry 0 rz 179.9 deg; joints [20.852, -38.703, 103.29, -156.968, 65.438, 170.546]
  MoveL 664 to (193.55, 220.92, -20.05) mm, rotated rx -180 ry 0 rz 179.9 deg; joints [20.842, -38.71, 103.307, -156.98, 65.445, 170.554]
  MoveL 665 to (193.48, 221.18, -20.05) mm, rotated rx -180 ry 0 rz 179.9 deg; joints [20.834, -38.717, 103.322, -156.99, 65.452, 170.561]
  MoveL 666 to (193.39, 221.43, -20.05) mm, rotated rx -180 ry 0 rz 179.9 deg; joints [20.826, -38.723, 103.338, -157.001, 65.459, 170.568]
  MoveL 667 to (193.29, 221.68, -20.05) mm, rotated rx -180 ry 0 rz 179.9 deg; joints [20.818, -38.731, 103.355, -157.011, 65.467, 170.576]
  MoveL 668 to (193.16, 221.93, -20.05) mm, rotated rx 180 ry 0 rz 179.9 deg; joints [20.811, -38.739, 103.374, -157.021, 65.476, 170.584]
  MoveL 669 to (193.02, 222.19, -20.05) mm, rotated rx -180 ry 0 rz 179.9 deg; joints [20.804, -38.747, 103.395, -157.03, 65.485, 170.592]
  MoveL 670 to (192.86, 222.44, -20.05) mm, rotated rx 180 ry 0 rz 179.9 deg; joints [20.797, -38.757, 103.417, -157.04, 65.496, 170.601]
  MoveL 671 to (192.68, 222.69, -20.05) mm, rotated rx 180 ry 0 rz 179.9 deg; joints [20.79, -38.767, 103.441, -157.05, 65.508, 170.609]
  MoveL 672 to (192.48, 222.94, -20.05) mm, rotated rx 180 ry 0 rz 179.9 deg; joints [20.784, -38.778, 103.467, -157.059, 65.521, 170.619]
  MoveL 673 to (192.27, 223.16, -20.05) mm, rotated rx 180 ry 0 rz 179.9 deg; joints [20.779, -38.789, 103.492, -157.067, 65.533, 170.627]
  MoveL 674 to (192.04, 223.38, -20.05) mm, rotated rx 180 ry 0 rz 179.9 deg; joints [20.774, -38.801, 103.519, -157.075, 65.547, 170.635]
  MoveL 675 to (191.79, 223.59, -20.05) mm, rotated rx 180 ry 0 rz 179.9 deg; joints [20.77, -38.813, 103.548, -157.082, 65.561, 170.644]
